(* Logix 5000 project; controller reports 1756-L63 rev 20.11; software revision 20.04; part 40 of 52 *)

        [82].log_data[53].total := -6932.722, [82].log_data[53].time := 3600.0, [82].log_data[53].minminute := 24, [82].log_data[53].maxminute := 3, [82].log_data[53].valid := 1, [82].log_data[54].max := 0.5155, [82].log_data[54].total := 1254.2913, [82].log_data[54].time := 3600.0, [82].log_data[54].minminute := 8, [82].log_data[54].maxminute := 9, [82].log_data[54].valid := 1, [82].log_data[55].max := 0.52349997, [82].log_data[55].total := 1217.507, [82].log_data[55].time := 3600.0, [82].log_data[55].minminute := 1, [82].log_data[55].maxminute := 24, [82].log_data[55].valid := 1, [82].log_data[56].min := 0.159696, [82].log_data[56].max := 0.16024561, [82].log_data[56].total := 575.79816, [82].log_data[56].time := 3600.0, [82].log_data[56].minminute := 6, [82].log_data[56].maxminute := 3, [82].log_data[56].valid := 1, [82].log_data[57].min := 0.24818413, [82].log_data[57].max := 0.2500293, [82].log_data[57].total := 894.9429, [82].log_data[57].time := 3600.0, [82].log_data[57].minminute := 17, [82].log_data[57].maxminute := 1, [82].log_data[57].valid := 1, [82].log_data[58].time := 3600.0, [82].log_data[58].valid := 1, [82].log_data[59].time := 3600.0, [82].log_data[59].valid := 1, [82].log_data[60].valid := 1, [82].log_data[61].valid := 1, [82].log_data[62].valid := 1, [82].log_data[63].valid := 1, [82].log_data[64].valid := 1, [82].log_data[65].valid := 1, [82].log_data[66].valid := 1, [82].log_data[67].valid := 1, [82].log_data[68].valid := 1, [82].log_data[69].valid := 1, [82].log_data[70].valid := 1, [82].log_data[71].valid := 1, [82].log_data[72].valid := 1, [82].log_data[73].valid := 1, [82].log_data[74].valid := 1, [82].log_data[75].valid := 1, [82].log_data[76].valid := 1, [82].log_data[77].valid := 1, [82].log_data[78].valid := 1, [82].log_data[79].valid := 1, [82].log_data[80].valid := 1, [82].log_data[81].valid := 1, [82].log_data[82].valid := 1, [82].log_data[83].valid := 1, [82].log_data[84].valid := 1,
        [82].log_data[85].valid := 1, [82].log_data[86].valid := 1, [82].log_data[87].valid := 1, [82].log_data[88].valid := 1, [82].log_data[89].valid := 1, [82].log_data[90].valid := 1, [82].log_data[91].valid := 1, [82].log_data[92].valid := 1, [82].log_data[93].valid := 1, [82].log_data[94].valid := 1, [82].log_data[95].valid := 1, [82].log_data[96].valid := 1, [82].log_data[97].valid := 1, [82].log_data[98].valid := 1, [82].log_data[99].valid := 1, [82].log_data[100].valid := 1, [82].log_data[101].valid := 1, [82].log_data[102].valid := 1, [82].log_data[103].valid := 1, [82].log_data[104].valid := 1, [82].log_data[105].valid := 1, [82].log_data[106].valid := 1, [82].log_data[107].valid := 1, [82].log_data[108].valid := 1, [82].log_data[109].valid := 1, [82].log_data[110].valid := 1, [82].log_data[111].valid := 1, [82].log_data[112].valid := 1, [82].log_data[113].valid := 1, [82].log_data[114].valid := 1, [82].log_data[115].valid := 1, [82].log_data[116].valid := 1, [82].log_data[117].valid := 1, [82].log_data[118].valid := 1, [82].log_data[119].valid := 1, [82].log_data[120].valid := 1, [82].log_data[121].valid := 1, [82].log_data[122].valid := 1, [82].log_data[123].valid := 1, [82].log_data[124].valid := 1, [82].time.Year := 2023, [82].time.Month := 1, [82].time.Day := 16, [82].time.Hour := 13, [82].time.Minute := 59, [82].time.Second := 59, [83].log_data[0].min := 1.0, [83].log_data[0].max := 1.0, [83].log_data[0].total := 3600.0, [83].log_data[0].time := 3600.0, [83].log_data[0].valid := 1, [83].log_data[1].max := 1.0, [83].log_data[1].total := 542.0, [83].log_data[1].time := 3600.0, [83].log_data[1].maxminute := 41, [83].log_data[1].valid := 1, [83].log_data[2].max := 1.0, [83].log_data[2].total := 538.5, [83].log_data[2].time := 3600.0, [83].log_data[2].maxminute := 41,
        [83].log_data[2].valid := 1, [83].log_data[3].time := 3600.0, [83].log_data[3].valid := 1, [83].log_data[4].time := 3600.0, [83].log_data[4].valid := 1, [83].log_data[5].max := 1.0, [83].log_data[5].total := 231.0, [83].log_data[5].time := 3600.0, [83].log_data[5].maxminute := 44, [83].log_data[5].valid := 1, [83].log_data[6].time := 3600.0, [83].log_data[6].valid := 1, [83].log_data[7].time := 3600.0, [83].log_data[7].valid := 1, [83].log_data[8].max := 1.0, [83].log_data[8].total := 1310.5, [83].log_data[8].time := 3600.0, [83].log_data[8].minminute := 10, [83].log_data[8].valid := 1, [83].log_data[9].max := 1.0, [83].log_data[9].total := 1307.0, [83].log_data[9].time := 3600.0, [83].log_data[9].minminute := 10, [83].log_data[9].valid := 1, [83].log_data[10].min := 1.0, [83].log_data[10].max := 1.0, [83].log_data[10].total := 3600.0, [83].log_data[10].time := 3600.0, [83].log_data[10].valid := 1, [83].log_data[11].time := 3600.0, [83].log_data[11].valid := 1, [83].log_data[12].min := 1.0, [83].log_data[12].max := 1.0, [83].log_data[12].total := 3600.0, [83].log_data[12].time := 3600.0, [83].log_data[12].valid := 1, [83].log_data[13].min := 1.0, [83].log_data[13].max := 1.0, [83].log_data[13].total := 3600.0, [83].log_data[13].time := 3600.0, [83].log_data[13].valid := 1, [83].log_data[14].time := 3600.0, [83].log_data[14].valid := 1, [83].log_data[15].time := 3600.0, [83].log_data[15].valid := 1, [83].log_data[16].time := 3600.0, [83].log_data[16].valid := 1, [83].log_data[17].min := 1.0, [83].log_data[17].max := 1.0, [83].log_data[17].total := 3600.0, [83].log_data[17].time := 3600.0, [83].log_data[17].valid := 1, [83].log_data[18].time := 3600.0, [83].log_data[18].valid := 1, [83].log_data[19].time := 3600.0, [83].log_data[19].valid := 1, [83].log_data[20].time := 3600.0, [83].log_data[20].valid := 1, [83].log_data[21].min := 1.0, [83].log_data[21].max := 1.0,
        [83].log_data[21].total := 3600.0, [83].log_data[21].time := 3600.0, [83].log_data[21].valid := 1, [83].log_data[22].time := 3600.0, [83].log_data[22].valid := 1, [83].log_data[23].time := 3600.0, [83].log_data[23].valid := 1, [83].log_data[24].time := 3600.0, [83].log_data[24].valid := 1, [83].log_data[25].time := 3600.0, [83].log_data[25].valid := 1, [83].log_data[26].time := 3600.0, [83].log_data[26].valid := 1, [83].log_data[27].time := 3600.0, [83].log_data[27].valid := 1, [83].log_data[28].time := 3600.0, [83].log_data[28].valid := 1, [83].log_data[29].min := 1.0, [83].log_data[29].max := 1.0, [83].log_data[29].total := 3600.0, [83].log_data[29].time := 3600.0, [83].log_data[29].valid := 1, [83].log_data[30].min := 1.0, [83].log_data[30].max := 1.0, [83].log_data[30].total := 3600.0, [83].log_data[30].time := 3600.0, [83].log_data[30].valid := 1, [83].log_data[31].max := 1.0, [83].log_data[31].total := 1071.998, [83].log_data[31].time := 3600.0, [83].log_data[31].maxminute := 2, [83].log_data[31].valid := 1, [83].log_data[32].max := 1.0, [83].log_data[32].total := 57.749, [83].log_data[32].time := 3600.0, [83].log_data[32].valid := 1, [83].log_data[33].max := 1.0, [83].log_data[33].total := 974.5, [83].log_data[33].time := 3600.0, [83].log_data[33].maxminute := 10, [83].log_data[33].valid := 1, [83].log_data[34].max := 1.0, [83].log_data[34].total := 987.5, [83].log_data[34].time := 3600.0, [83].log_data[34].maxminute := 8, [83].log_data[34].valid := 1, [83].log_data[35].max := 1.0, [83].log_data[35].total := 538.998, [83].log_data[35].time := 3600.0, [83].log_data[35].maxminute := 6, [83].log_data[35].valid := 1, [83].log_data[36].max := 1.0, [83].log_data[36].total := 571.5, [83].log_data[36].time := 3600.0, [83].log_data[36].minminute := 5, [83].log_data[36].valid := 1, [83].log_data[37].max := 7.3565416, [83].log_data[37].total := 3456.338, [83].log_data[37].time := 3600.0, [83].log_data[37].maxminute := 44,
        [83].log_data[37].valid := 1, [83].log_data[38].time := 3600.0, [83].log_data[38].valid := 1, [83].log_data[39].min := 0.994824, [83].log_data[39].max := 1.0214411, [83].log_data[39].total := 3605.966, [83].log_data[39].time := 3600.0, [83].log_data[39].minminute := 3, [83].log_data[39].maxminute := 48, [83].log_data[39].valid := 1, [83].log_data[40].min := 7.574485, [83].log_data[40].max := 7.60224, [83].log_data[40].total := 27337.104, [83].log_data[40].time := 3600.0, [83].log_data[40].minminute := 29, [83].log_data[40].maxminute := 32, [83].log_data[40].valid := 1, [83].log_data[41].min := 0.02273633, [83].log_data[41].max := 0.035495363, [83].log_data[41].total := 89.72992, [83].log_data[41].time := 3600.0, [83].log_data[41].minminute := 20, [83].log_data[41].maxminute := 32, [83].log_data[41].valid := 1, [83].log_data[42].min := 2.291407, [83].log_data[42].max := 2.2964714, [83].log_data[42].total := 8258.98, [83].log_data[42].time := 3600.0, [83].log_data[42].minminute := 56, [83].log_data[42].maxminute := 28, [83].log_data[42].valid := 1, [83].log_data[43].min := -0.27999878, [83].log_data[43].max := -0.26000214, [83].log_data[43].total := -981.76685, [83].log_data[43].time := 3600.0, [83].log_data[43].maxminute := 2, [83].log_data[43].valid := 1, [83].log_data[44].min := -0.3199997, [83].log_data[44].max := -0.30000305, [83].log_data[44].total := -1089.0538, [83].log_data[44].time := 3600.0, [83].log_data[44].valid := 1, [83].log_data[45].time := 3600.0, [83].log_data[45].valid := 1, [83].log_data[46].time := 3600.0, [83].log_data[46].valid := 1, [83].log_data[47].time := 3600.0, [83].log_data[47].valid := 1, [83].log_data[48].min := 6.7179084, [83].log_data[48].max := 6.9322586, [83].log_data[48].total := 24380.49, [83].log_data[48].time := 3600.0, [83].log_data[48].minminute := 59, [83].log_data[48].maxminute := 50, [83].log_data[48].valid := 1, [83].log_data[49].min := 7.303773, [83].log_data[49].max := 9.598419, [83].log_data[49].total := 33269.867, [83].log_data[49].time := 3600.0, [83].log_data[49].minminute := 59,
        [83].log_data[49].maxminute := 5, [83].log_data[49].valid := 1, [83].log_data[50].min := 1.9989722, [83].log_data[50].max := 2.151373, [83].log_data[50].total := 7406.148, [83].log_data[50].time := 3600.0, [83].log_data[50].minminute := 10, [83].log_data[50].maxminute := 49, [83].log_data[50].valid := 1, [83].log_data[51].max := 3.127, [83].log_data[51].total := 2959.4797, [83].log_data[51].time := 3600.0, [83].log_data[51].maxminute := 10, [83].log_data[51].valid := 1, [83].log_data[52].min := -5.739998, [83].log_data[52].max := 0.11999512, [83].log_data[52].total := -8463.669, [83].log_data[52].time := 3600.0, [83].log_data[52].minminute := 49, [83].log_data[52].valid := 1, [83].log_data[53].min := -4.919998, [83].log_data[53].max := 0.30000305, [83].log_data[53].total := -7675.482, [83].log_data[53].time := 3600.0, [83].log_data[53].minminute := 49, [83].log_data[53].maxminute := 55, [83].log_data[53].valid := 1, [83].log_data[54].max := 0.56850004, [83].log_data[54].total := 446.67337, [83].log_data[54].time := 3600.0, [83].log_data[54].maxminute := 2, [83].log_data[54].valid := 1, [83].log_data[55].max := 0.543, [83].log_data[55].total := 438.6968, [83].log_data[55].time := 3600.0, [83].log_data[55].minminute := 5, [83].log_data[55].maxminute := 55, [83].log_data[55].valid := 1, [83].log_data[56].min := 0.15973525, [83].log_data[56].max := 0.16016708, [83].log_data[56].total := 575.74774, [83].log_data[56].time := 3600.0, [83].log_data[56].minminute := 12, [83].log_data[56].maxminute := 17, [83].log_data[56].valid := 1, [83].log_data[57].min := 0.24818413, [83].log_data[57].max := 0.24861601, [83].log_data[57].total := 894.0131, [83].log_data[57].time := 3600.0, [83].log_data[57].maxminute := 39, [83].log_data[57].valid := 1, [83].log_data[58].time := 3600.0, [83].log_data[58].valid := 1, [83].log_data[59].time := 3600.0, [83].log_data[59].valid := 1, [83].log_data[60].valid := 1, [83].log_data[61].valid := 1, [83].log_data[62].valid := 1, [83].log_data[63].valid := 1, [83].log_data[64].valid := 1,
        [83].log_data[65].valid := 1, [83].log_data[66].valid := 1, [83].log_data[67].valid := 1, [83].log_data[68].valid := 1, [83].log_data[69].valid := 1, [83].log_data[70].valid := 1, [83].log_data[71].valid := 1, [83].log_data[72].valid := 1, [83].log_data[73].valid := 1, [83].log_data[74].valid := 1, [83].log_data[75].valid := 1, [83].log_data[76].valid := 1, [83].log_data[77].valid := 1, [83].log_data[78].valid := 1, [83].log_data[79].valid := 1, [83].log_data[80].valid := 1, [83].log_data[81].valid := 1, [83].log_data[82].valid := 1, [83].log_data[83].valid := 1, [83].log_data[84].valid := 1, [83].log_data[85].valid := 1, [83].log_data[86].valid := 1, [83].log_data[87].valid := 1, [83].log_data[88].valid := 1, [83].log_data[89].valid := 1, [83].log_data[90].valid := 1, [83].log_data[91].valid := 1, [83].log_data[92].valid := 1, [83].log_data[93].valid := 1, [83].log_data[94].valid := 1, [83].log_data[95].valid := 1, [83].log_data[96].valid := 1, [83].log_data[97].valid := 1, [83].log_data[98].valid := 1, [83].log_data[99].valid := 1, [83].log_data[100].valid := 1, [83].log_data[101].valid := 1, [83].log_data[102].valid := 1, [83].log_data[103].valid := 1, [83].log_data[104].valid := 1, [83].log_data[105].valid := 1, [83].log_data[106].valid := 1, [83].log_data[107].valid := 1, [83].log_data[108].valid := 1, [83].log_data[109].valid := 1, [83].log_data[110].valid := 1, [83].log_data[111].valid := 1, [83].log_data[112].valid := 1, [83].log_data[113].valid := 1, [83].log_data[114].valid := 1, [83].log_data[115].valid := 1, [83].log_data[116].valid := 1, [83].log_data[117].valid := 1, [83].log_data[118].valid := 1, [83].log_data[119].valid := 1, [83].log_data[120].valid := 1, [83].log_data[121].valid := 1, [83].log_data[122].valid := 1, [83].log_data[123].valid := 1, [83].log_data[124].valid := 1,
        [83].time.Year := 2023, [83].time.Month := 1, [83].time.Day := 16, [83].time.Hour := 14, [83].time.Minute := 59, [83].time.Second := 59, [84].log_data[0].min := 1.0, [84].log_data[0].max := 1.0, [84].log_data[0].total := 3600.0, [84].log_data[0].time := 3600.0, [84].log_data[0].valid := 1, [84].log_data[1].time := 3600.0, [84].log_data[1].valid := 1, [84].log_data[2].time := 3600.0, [84].log_data[2].valid := 1, [84].log_data[3].time := 3600.0, [84].log_data[3].valid := 1, [84].log_data[4].time := 3600.0, [84].log_data[4].valid := 1, [84].log_data[5].time := 3600.0, [84].log_data[5].valid := 1, [84].log_data[6].time := 3600.0, [84].log_data[6].valid := 1, [84].log_data[7].time := 3600.0, [84].log_data[7].valid := 1, [84].log_data[8].max := 1.0, [84].log_data[8].total := 322.251, [84].log_data[8].time := 3600.0, [84].log_data[8].minminute := 5, [84].log_data[8].valid := 1, [84].log_data[9].max := 1.0, [84].log_data[9].total := 322.251, [84].log_data[9].time := 3600.0, [84].log_data[9].minminute := 5, [84].log_data[9].valid := 1, [84].log_data[10].min := 1.0, [84].log_data[10].max := 1.0, [84].log_data[10].total := 3600.0, [84].log_data[10].time := 3600.0, [84].log_data[10].valid := 1, [84].log_data[11].time := 3600.0, [84].log_data[11].valid := 1, [84].log_data[12].min := 1.0, [84].log_data[12].max := 1.0, [84].log_data[12].total := 3600.0, [84].log_data[12].time := 3600.0, [84].log_data[12].valid := 1, [84].log_data[13].min := 1.0, [84].log_data[13].max := 1.0, [84].log_data[13].total := 3600.0, [84].log_data[13].time := 3600.0, [84].log_data[13].valid := 1, [84].log_data[14].time := 3600.0, [84].log_data[14].valid := 1, [84].log_data[15].time := 3600.0, [84].log_data[15].valid := 1, [84].log_data[16].time := 3600.0, [84].log_data[16].valid := 1, [84].log_data[17].min := 1.0, [84].log_data[17].max := 1.0,
        [84].log_data[17].total := 3600.0, [84].log_data[17].time := 3600.0, [84].log_data[17].valid := 1, [84].log_data[18].time := 3600.0, [84].log_data[18].valid := 1, [84].log_data[19].time := 3600.0, [84].log_data[19].valid := 1, [84].log_data[20].time := 3600.0, [84].log_data[20].valid := 1, [84].log_data[21].min := 1.0, [84].log_data[21].max := 1.0, [84].log_data[21].total := 3600.0, [84].log_data[21].time := 3600.0, [84].log_data[21].valid := 1, [84].log_data[22].time := 3600.0, [84].log_data[22].valid := 1, [84].log_data[23].time := 3600.0, [84].log_data[23].valid := 1, [84].log_data[24].time := 3600.0, [84].log_data[24].valid := 1, [84].log_data[25].time := 3600.0, [84].log_data[25].valid := 1, [84].log_data[26].time := 3600.0, [84].log_data[26].valid := 1, [84].log_data[27].time := 3600.0, [84].log_data[27].valid := 1, [84].log_data[28].time := 3600.0, [84].log_data[28].valid := 1, [84].log_data[29].min := 1.0, [84].log_data[29].max := 1.0, [84].log_data[29].total := 3600.0, [84].log_data[29].time := 3600.0, [84].log_data[29].valid := 1, [84].log_data[30].min := 1.0, [84].log_data[30].max := 1.0, [84].log_data[30].total := 3600.0, [84].log_data[30].time := 3600.0, [84].log_data[30].valid := 1, [84].log_data[31].time := 3600.0, [84].log_data[31].valid := 1, [84].log_data[32].max := 1.0, [84].log_data[32].total := 238.749, [84].log_data[32].time := 3600.0, [84].log_data[32].maxminute := 1, [84].log_data[32].valid := 1, [84].log_data[33].time := 3600.0, [84].log_data[33].valid := 1, [84].log_data[34].time := 3600.0, [84].log_data[34].valid := 1, [84].log_data[35].max := 1.0, [84].log_data[35].total := 276.0, [84].log_data[35].time := 3600.0, [84].log_data[35].minminute := 4, [84].log_data[35].valid := 1, [84].log_data[36].time := 3600.0, [84].log_data[36].valid := 1, [84].log_data[37].time := 3600.0, [84].log_data[37].valid := 1, [84].log_data[38].time := 3600.0, [84].log_data[38].valid := 1,
        [84].log_data[39].min := 0.99494183, [84].log_data[39].max := 1.0055416, [84].log_data[39].total := 3602.3838, [84].log_data[39].time := 3600.0, [84].log_data[39].minminute := 16, [84].log_data[39].maxminute := 46, [84].log_data[39].valid := 1, [84].log_data[40].min := 7.5816298, [84].log_data[40].max := 7.604989, [84].log_data[40].total := 27343.059, [84].log_data[40].time := 3600.0, [84].log_data[40].minminute := 26, [84].log_data[40].maxminute := 37, [84].log_data[40].valid := 1, [84].log_data[41].min := 0.02273633, [84].log_data[41].max := 0.030195557, [84].log_data[41].total := 87.1149, [84].log_data[41].time := 3600.0, [84].log_data[41].minminute := 1, [84].log_data[41].maxminute := 57, [84].log_data[41].valid := 1, [84].log_data[42].min := 2.291525, [84].log_data[42].max := 2.2963536, [84].log_data[42].total := 8259.134, [84].log_data[42].time := 3600.0, [84].log_data[42].minminute := 10, [84].log_data[42].maxminute := 47, [84].log_data[42].valid := 1, [84].log_data[43].min := -0.27999878, [84].log_data[43].max := -0.26000214, [84].log_data[43].total := -936.00824, [84].log_data[43].time := 3600.0, [84].log_data[43].valid := 1, [84].log_data[44].min := -0.30000305, [84].log_data[44].max := -0.27999878, [84].log_data[44].total := -1061.0931, [84].log_data[44].time := 3600.0, [84].log_data[44].maxminute := 5, [84].log_data[44].valid := 1, [84].log_data[45].time := 3600.0, [84].log_data[45].valid := 1, [84].log_data[46].time := 3600.0, [84].log_data[46].valid := 1, [84].log_data[47].time := 3600.0, [84].log_data[47].valid := 1, [84].log_data[48].min := 6.5678625, [84].log_data[48].max := 6.7181826, [84].log_data[48].total := 23808.375, [84].log_data[48].time := 3600.0, [84].log_data[48].minminute := 18, [84].log_data[48].valid := 1, [84].log_data[49].min := 6.593787, [84].log_data[49].max := 9.412138, [84].log_data[49].total := 28587.87, [84].log_data[49].time := 3600.0, [84].log_data[49].minminute := 17, [84].log_data[49].maxminute := 59, [84].log_data[49].valid := 1, [84].log_data[50].min := 1.9986188, [84].log_data[50].max := 2.109445,
        [84].log_data[50].total := 7530.9287, [84].log_data[50].time := 3600.0, [84].log_data[50].minminute := 5, [84].log_data[50].maxminute := 57, [84].log_data[50].valid := 1, [84].log_data[51].time := 3600.0, [84].log_data[51].valid := 1, [84].log_data[52].min := -2.9199982, [84].log_data[52].max := 0.11999512, [84].log_data[52].total := -5281.0723, [84].log_data[52].time := 3600.0, [84].log_data[52].minminute := 1, [84].log_data[52].valid := 1, [84].log_data[53].min := -2.4000015, [84].log_data[53].max := 0.22000122, [84].log_data[53].total := -5018.0986, [84].log_data[53].time := 3600.0, [84].log_data[53].minminute := 4, [84].log_data[53].maxminute := 5, [84].log_data[53].valid := 1, [84].log_data[54].max := 0.523, [84].log_data[54].total := 93.84478, [84].log_data[54].time := 3600.0, [84].log_data[54].maxminute := 1, [84].log_data[54].valid := 1, [84].log_data[55].max := 0.4465, [84].log_data[55].total := 110.74925, [84].log_data[55].time := 3600.0, [84].log_data[55].minminute := 4, [84].log_data[55].maxminute := 4, [84].log_data[55].valid := 1, [84].log_data[56].min := 0.15973525, [84].log_data[56].max := 0.16012783, [84].log_data[56].total := 575.5827, [84].log_data[56].time := 3600.0, [84].log_data[56].minminute := 19, [84].log_data[56].maxminute := 1, [84].log_data[56].valid := 1, [84].log_data[57].min := 0.24826264, [84].log_data[57].max := 0.24869452, [84].log_data[57].total := 894.43835, [84].log_data[57].time := 3600.0, [84].log_data[57].minminute := 23, [84].log_data[57].maxminute := 37, [84].log_data[57].valid := 1, [84].log_data[58].time := 3600.0, [84].log_data[58].valid := 1, [84].log_data[59].time := 3600.0, [84].log_data[59].valid := 1, [84].log_data[60].valid := 1, [84].log_data[61].valid := 1, [84].log_data[62].valid := 1, [84].log_data[63].valid := 1, [84].log_data[64].valid := 1, [84].log_data[65].valid := 1, [84].log_data[66].valid := 1, [84].log_data[67].valid := 1, [84].log_data[68].valid := 1, [84].log_data[69].valid := 1, [84].log_data[70].valid := 1,
        [84].log_data[71].valid := 1, [84].log_data[72].valid := 1, [84].log_data[73].valid := 1, [84].log_data[74].valid := 1, [84].log_data[75].valid := 1, [84].log_data[76].valid := 1, [84].log_data[77].valid := 1, [84].log_data[78].valid := 1, [84].log_data[79].valid := 1, [84].log_data[80].valid := 1, [84].log_data[81].valid := 1, [84].log_data[82].valid := 1, [84].log_data[83].valid := 1, [84].log_data[84].valid := 1, [84].log_data[85].valid := 1, [84].log_data[86].valid := 1, [84].log_data[87].valid := 1, [84].log_data[88].valid := 1, [84].log_data[89].valid := 1, [84].log_data[90].valid := 1, [84].log_data[91].valid := 1, [84].log_data[92].valid := 1, [84].log_data[93].valid := 1, [84].log_data[94].valid := 1, [84].log_data[95].valid := 1, [84].log_data[96].valid := 1, [84].log_data[97].valid := 1, [84].log_data[98].valid := 1, [84].log_data[99].valid := 1, [84].log_data[100].valid := 1, [84].log_data[101].valid := 1, [84].log_data[102].valid := 1, [84].log_data[103].valid := 1, [84].log_data[104].valid := 1, [84].log_data[105].valid := 1, [84].log_data[106].valid := 1, [84].log_data[107].valid := 1, [84].log_data[108].valid := 1, [84].log_data[109].valid := 1, [84].log_data[110].valid := 1, [84].log_data[111].valid := 1, [84].log_data[112].valid := 1, [84].log_data[113].valid := 1, [84].log_data[114].valid := 1, [84].log_data[115].valid := 1, [84].log_data[116].valid := 1, [84].log_data[117].valid := 1, [84].log_data[118].valid := 1, [84].log_data[119].valid := 1, [84].log_data[120].valid := 1, [84].log_data[121].valid := 1, [84].log_data[122].valid := 1, [84].log_data[123].valid := 1, [84].log_data[124].valid := 1, [84].time.Year := 2023, [84].time.Month := 1, [84].time.Day := 16, [84].time.Hour := 15, [84].time.Minute := 59, [84].time.Second := 59,
        [85].log_data[0].min := 1.0, [85].log_data[0].max := 1.0, [85].log_data[0].total := 3600.0, [85].log_data[0].time := 3600.0, [85].log_data[0].valid := 1, [85].log_data[1].max := 1.0, [85].log_data[1].total := 541.5, [85].log_data[1].time := 3600.0, [85].log_data[1].maxminute := 47, [85].log_data[1].valid := 1, [85].log_data[2].max := 1.0, [85].log_data[2].total := 538.0, [85].log_data[2].time := 3600.0, [85].log_data[2].maxminute := 47, [85].log_data[2].valid := 1, [85].log_data[3].time := 3600.0, [85].log_data[3].valid := 1, [85].log_data[4].time := 3600.0, [85].log_data[4].valid := 1, [85].log_data[5].max := 1.0, [85].log_data[5].total := 244.5, [85].log_data[5].time := 3600.0, [85].log_data[5].maxminute := 49, [85].log_data[5].valid := 1, [85].log_data[6].time := 3600.0, [85].log_data[6].valid := 1, [85].log_data[7].time := 3600.0, [85].log_data[7].valid := 1, [85].log_data[8].max := 1.0, [85].log_data[8].total := 508.749, [85].log_data[8].time := 3600.0, [85].log_data[8].maxminute := 51, [85].log_data[8].valid := 1, [85].log_data[9].max := 1.0, [85].log_data[9].total := 505.249, [85].log_data[9].time := 3600.0, [85].log_data[9].maxminute := 51, [85].log_data[9].valid := 1, [85].log_data[10].min := 1.0, [85].log_data[10].max := 1.0, [85].log_data[10].total := 3600.0, [85].log_data[10].time := 3600.0, [85].log_data[10].valid := 1, [85].log_data[11].time := 3600.0, [85].log_data[11].valid := 1, [85].log_data[12].min := 1.0, [85].log_data[12].max := 1.0, [85].log_data[12].total := 3600.0, [85].log_data[12].time := 3600.0, [85].log_data[12].valid := 1, [85].log_data[13].min := 1.0, [85].log_data[13].max := 1.0, [85].log_data[13].total := 3600.0, [85].log_data[13].time := 3600.0, [85].log_data[13].valid := 1, [85].log_data[14].time := 3600.0, [85].log_data[14].valid := 1, [85].log_data[15].time := 3600.0, [85].log_data[15].valid := 1, [85].log_data[16].time := 3600.0,
        [85].log_data[16].valid := 1, [85].log_data[17].min := 1.0, [85].log_data[17].max := 1.0, [85].log_data[17].total := 3600.0, [85].log_data[17].time := 3600.0, [85].log_data[17].valid := 1, [85].log_data[18].time := 3600.0, [85].log_data[18].valid := 1, [85].log_data[19].time := 3600.0, [85].log_data[19].valid := 1, [85].log_data[20].time := 3600.0, [85].log_data[20].valid := 1, [85].log_data[21].min := 1.0, [85].log_data[21].max := 1.0, [85].log_data[21].total := 3600.0, [85].log_data[21].time := 3600.0, [85].log_data[21].valid := 1, [85].log_data[22].time := 3600.0, [85].log_data[22].valid := 1, [85].log_data[23].time := 3600.0, [85].log_data[23].valid := 1, [85].log_data[24].time := 3600.0, [85].log_data[24].valid := 1, [85].log_data[25].time := 3600.0, [85].log_data[25].valid := 1, [85].log_data[26].time := 3600.0, [85].log_data[26].valid := 1, [85].log_data[27].time := 3600.0, [85].log_data[27].valid := 1, [85].log_data[28].time := 3600.0, [85].log_data[28].valid := 1, [85].log_data[29].min := 1.0, [85].log_data[29].max := 1.0, [85].log_data[29].total := 3600.0, [85].log_data[29].time := 3600.0, [85].log_data[29].valid := 1, [85].log_data[30].min := 1.0, [85].log_data[30].max := 1.0, [85].log_data[30].total := 3600.0, [85].log_data[30].time := 3600.0, [85].log_data[30].valid := 1, [85].log_data[31].max := 1.0, [85].log_data[31].total := 304.249, [85].log_data[31].time := 3600.0, [85].log_data[31].maxminute := 51, [85].log_data[31].valid := 1, [85].log_data[32].max := 1.0, [85].log_data[32].total := 109.249, [85].log_data[32].time := 3600.0, [85].log_data[32].maxminute := 58, [85].log_data[32].valid := 1, [85].log_data[33].time := 3600.0, [85].log_data[33].valid := 1, [85].log_data[34].time := 3600.0, [85].log_data[34].valid := 1, [85].log_data[35].time := 3600.0, [85].log_data[35].valid := 1, [85].log_data[36].max := 1.0, [85].log_data[36].total := 498.249, [85].log_data[36].time := 3600.0,
        [85].log_data[36].maxminute := 51, [85].log_data[36].valid := 1, [85].log_data[37].max := 7.6030836, [85].log_data[37].total := 3563.115, [85].log_data[37].time := 3600.0, [85].log_data[37].maxminute := 49, [85].log_data[37].valid := 1, [85].log_data[38].time := 3600.0, [85].log_data[38].valid := 1, [85].log_data[39].min := 0.994824, [85].log_data[39].max := 1.0213233, [85].log_data[39].total := 3607.2905, [85].log_data[39].time := 3600.0, [85].log_data[39].minminute := 13, [85].log_data[39].maxminute := 54, [85].log_data[39].valid := 1, [85].log_data[40].min := 7.5802555, [85].log_data[40].max := 7.603339, [85].log_data[40].total := 27341.73, [85].log_data[40].time := 3600.0, [85].log_data[40].minminute := 26, [85].log_data[40].maxminute := 31, [85].log_data[40].valid := 1, [85].log_data[41].min := 0.02273633, [85].log_data[41].max := 0.036476806, [85].log_data[41].total := 93.75936, [85].log_data[41].time := 3600.0, [85].log_data[41].minminute := 19, [85].log_data[41].maxminute := 12, [85].log_data[41].valid := 1, [85].log_data[42].min := 2.291525, [85].log_data[42].max := 2.2964714, [85].log_data[42].total := 8259.261, [85].log_data[42].time := 3600.0, [85].log_data[42].minminute := 7, [85].log_data[42].maxminute := 41, [85].log_data[42].valid := 1, [85].log_data[43].min := -0.26000214, [85].log_data[43].max := -0.23999786, [85].log_data[43].total := -935.90826, [85].log_data[43].time := 3600.0, [85].log_data[43].maxminute := 1, [85].log_data[43].valid := 1, [85].log_data[44].min := -0.30000305, [85].log_data[44].max := -0.27999878, [85].log_data[44].total := -1013.5552, [85].log_data[44].time := 3600.0, [85].log_data[44].valid := 1, [85].log_data[45].time := 3600.0, [85].log_data[45].valid := 1, [85].log_data[46].time := 3600.0, [85].log_data[46].valid := 1, [85].log_data[47].time := 3600.0, [85].log_data[47].valid := 1, [85].log_data[48].min := 6.6335416, [85].log_data[48].max := 6.9078, [85].log_data[48].total := 24063.035, [85].log_data[48].time := 3600.0, [85].log_data[48].maxminute := 56, [85].log_data[48].valid := 1,
        [85].log_data[49].min := 8.170596, [85].log_data[49].max := 9.692444, [85].log_data[49].total := 34133.863, [85].log_data[49].time := 3600.0, [85].log_data[49].minminute := 59, [85].log_data[49].maxminute := 49, [85].log_data[49].valid := 1, [85].log_data[50].min := 2.0683415, [85].log_data[50].max := 2.1509018, [85].log_data[50].total := 7587.8726, [85].log_data[50].time := 3600.0, [85].log_data[50].minminute := 54, [85].log_data[50].maxminute := 51, [85].log_data[50].valid := 1, [85].log_data[51].time := 3600.0, [85].log_data[51].valid := 1, [85].log_data[52].min := -4.3199997, [85].log_data[52].max := 0.11999512, [85].log_data[52].total := -5856.0786, [85].log_data[52].time := 3600.0, [85].log_data[52].minminute := 51, [85].log_data[52].maxminute := 56, [85].log_data[52].valid := 1, [85].log_data[53].min := -4.040001, [85].log_data[53].max := -1.4400024, [85].log_data[53].total := -5783.3413, [85].log_data[53].time := 3600.0, [85].log_data[53].minminute := 51, [85].log_data[53].valid := 1, [85].log_data[54].max := 0.508, [85].log_data[54].total := 161.4602, [85].log_data[54].time := 3600.0, [85].log_data[54].maxminute := 51, [85].log_data[54].valid := 1, [85].log_data[55].max := 0.5005, [85].log_data[55].total := 197.12991, [85].log_data[55].time := 3600.0, [85].log_data[55].maxminute := 51, [85].log_data[55].valid := 1, [85].log_data[56].min := 0.15961748, [85].log_data[56].max := 0.16012783, [85].log_data[56].total := 575.4132, [85].log_data[56].time := 3600.0, [85].log_data[56].minminute := 45, [85].log_data[56].maxminute := 49, [85].log_data[56].valid := 1, [85].log_data[57].min := 0.24838047, [85].log_data[57].max := 0.2488123, [85].log_data[57].total := 894.79694, [85].log_data[57].time := 3600.0, [85].log_data[57].minminute := 3, [85].log_data[57].maxminute := 25, [85].log_data[57].valid := 1, [85].log_data[58].time := 3600.0, [85].log_data[58].valid := 1, [85].log_data[59].time := 3600.0, [85].log_data[59].valid := 1, [85].log_data[60].valid := 1, [85].log_data[61].valid := 1, [85].log_data[62].valid := 1,
        [85].log_data[63].valid := 1, [85].log_data[64].valid := 1, [85].log_data[65].valid := 1, [85].log_data[66].valid := 1, [85].log_data[67].valid := 1, [85].log_data[68].valid := 1, [85].log_data[69].valid := 1, [85].log_data[70].valid := 1, [85].log_data[71].valid := 1, [85].log_data[72].valid := 1, [85].log_data[73].valid := 1, [85].log_data[74].valid := 1, [85].log_data[75].valid := 1, [85].log_data[76].valid := 1, [85].log_data[77].valid := 1, [85].log_data[78].valid := 1, [85].log_data[79].valid := 1, [85].log_data[80].valid := 1, [85].log_data[81].valid := 1, [85].log_data[82].valid := 1, [85].log_data[83].valid := 1, [85].log_data[84].valid := 1, [85].log_data[85].valid := 1, [85].log_data[86].valid := 1, [85].log_data[87].valid := 1, [85].log_data[88].valid := 1, [85].log_data[89].valid := 1, [85].log_data[90].valid := 1, [85].log_data[91].valid := 1, [85].log_data[92].valid := 1, [85].log_data[93].valid := 1, [85].log_data[94].valid := 1, [85].log_data[95].valid := 1, [85].log_data[96].valid := 1, [85].log_data[97].valid := 1, [85].log_data[98].valid := 1, [85].log_data[99].valid := 1, [85].log_data[100].valid := 1, [85].log_data[101].valid := 1, [85].log_data[102].valid := 1, [85].log_data[103].valid := 1, [85].log_data[104].valid := 1, [85].log_data[105].valid := 1, [85].log_data[106].valid := 1, [85].log_data[107].valid := 1, [85].log_data[108].valid := 1, [85].log_data[109].valid := 1, [85].log_data[110].valid := 1, [85].log_data[111].valid := 1, [85].log_data[112].valid := 1, [85].log_data[113].valid := 1, [85].log_data[114].valid := 1, [85].log_data[115].valid := 1, [85].log_data[116].valid := 1, [85].log_data[117].valid := 1, [85].log_data[118].valid := 1, [85].log_data[119].valid := 1, [85].log_data[120].valid := 1, [85].log_data[121].valid := 1, [85].log_data[122].valid := 1,
        [85].log_data[123].valid := 1, [85].log_data[124].valid := 1, [85].time.Year := 2023, [85].time.Month := 1, [85].time.Day := 16, [85].time.Hour := 16, [85].time.Minute := 59, [85].time.Second := 59, [86].log_data[0].min := 1.0, [86].log_data[0].max := 1.0, [86].log_data[0].total := 3600.0, [86].log_data[0].time := 3600.0, [86].log_data[0].valid := 1, [86].log_data[1].time := 3600.0, [86].log_data[1].valid := 1, [86].log_data[2].time := 3600.0, [86].log_data[2].valid := 1, [86].log_data[3].time := 3600.0, [86].log_data[3].valid := 1, [86].log_data[4].time := 3600.0, [86].log_data[4].valid := 1, [86].log_data[5].time := 3600.0, [86].log_data[5].valid := 1, [86].log_data[6].time := 3600.0, [86].log_data[6].valid := 1, [86].log_data[7].time := 3600.0, [86].log_data[7].valid := 1, [86].log_data[8].min := 1.0, [86].log_data[8].max := 1.0, [86].log_data[8].total := 3600.0, [86].log_data[8].time := 3600.0, [86].log_data[8].valid := 1, [86].log_data[9].min := 1.0, [86].log_data[9].max := 1.0, [86].log_data[9].total := 3600.0, [86].log_data[9].time := 3600.0, [86].log_data[9].valid := 1, [86].log_data[10].min := 1.0, [86].log_data[10].max := 1.0, [86].log_data[10].total := 3600.0, [86].log_data[10].time := 3600.0, [86].log_data[10].valid := 1, [86].log_data[11].time := 3600.0, [86].log_data[11].valid := 1, [86].log_data[12].min := 1.0, [86].log_data[12].max := 1.0, [86].log_data[12].total := 3600.0, [86].log_data[12].time := 3600.0, [86].log_data[12].valid := 1, [86].log_data[13].min := 1.0, [86].log_data[13].max := 1.0, [86].log_data[13].total := 3600.0, [86].log_data[13].time := 3600.0, [86].log_data[13].valid := 1, [86].log_data[14].time := 3600.0, [86].log_data[14].valid := 1, [86].log_data[15].time := 3600.0, [86].log_data[15].valid := 1, [86].log_data[16].time := 3600.0, [86].log_data[16].valid := 1,
        [86].log_data[17].min := 1.0, [86].log_data[17].max := 1.0, [86].log_data[17].total := 3600.0, [86].log_data[17].time := 3600.0, [86].log_data[17].valid := 1, [86].log_data[18].time := 3600.0, [86].log_data[18].valid := 1, [86].log_data[19].time := 3600.0, [86].log_data[19].valid := 1, [86].log_data[20].time := 3600.0, [86].log_data[20].valid := 1, [86].log_data[21].min := 1.0, [86].log_data[21].max := 1.0, [86].log_data[21].total := 3600.0, [86].log_data[21].time := 3600.0, [86].log_data[21].valid := 1, [86].log_data[22].time := 3600.0, [86].log_data[22].valid := 1, [86].log_data[23].time := 3600.0, [86].log_data[23].valid := 1, [86].log_data[24].time := 3600.0, [86].log_data[24].valid := 1, [86].log_data[25].time := 3600.0, [86].log_data[25].valid := 1, [86].log_data[26].time := 3600.0, [86].log_data[26].valid := 1, [86].log_data[27].time := 3600.0, [86].log_data[27].valid := 1, [86].log_data[28].time := 3600.0, [86].log_data[28].valid := 1, [86].log_data[29].min := 1.0, [86].log_data[29].max := 1.0, [86].log_data[29].total := 3600.0, [86].log_data[29].time := 3600.0, [86].log_data[29].valid := 1, [86].log_data[30].min := 1.0, [86].log_data[30].max := 1.0, [86].log_data[30].total := 3600.0, [86].log_data[30].time := 3600.0, [86].log_data[30].valid := 1, [86].log_data[31].max := 1.0, [86].log_data[31].total := 1629.7471, [86].log_data[31].time := 3600.0, [86].log_data[31].maxminute := 8, [86].log_data[31].valid := 1, [86].log_data[32].max := 1.0, [86].log_data[32].total := 1520.749, [86].log_data[32].time := 3600.0, [86].log_data[32].minminute := 7, [86].log_data[32].valid := 1, [86].log_data[33].time := 3600.0, [86].log_data[33].valid := 1, [86].log_data[34].time := 3600.0, [86].log_data[34].valid := 1, [86].log_data[35].max := 1.0, [86].log_data[35].total := 1629.7471, [86].log_data[35].time := 3600.0, [86].log_data[35].maxminute := 2, [86].log_data[35].valid := 1, [86].log_data[36].max := 1.0,
        [86].log_data[36].total := 1440.498, [86].log_data[36].time := 3600.0, [86].log_data[36].valid := 1, [86].log_data[37].time := 3600.0, [86].log_data[37].valid := 1, [86].log_data[38].time := 3600.0, [86].log_data[38].valid := 1, [86].log_data[39].min := 0.9934107, [86].log_data[39].max := 1.0044814, [86].log_data[39].total := 3599.212, [86].log_data[39].time := 3600.0, [86].log_data[39].minminute := 44, [86].log_data[39].maxminute := 47, [86].log_data[39].valid := 1, [86].log_data[40].min := 7.5871253, [86].log_data[40].max := 7.603339, [86].log_data[40].total := 27345.953, [86].log_data[40].time := 3600.0, [86].log_data[40].minminute := 21, [86].log_data[40].maxminute := 28, [86].log_data[40].valid := 1, [86].log_data[41].min := 0.022540038, [86].log_data[41].max := 0.028232668, [86].log_data[41].total := 83.212074, [86].log_data[41].time := 3600.0, [86].log_data[41].minminute := 17, [86].log_data[41].maxminute := 1, [86].log_data[41].valid := 1, [86].log_data[42].min := 2.2916427, [86].log_data[42].max := 2.2963536, [86].log_data[42].total := 8259.18, [86].log_data[42].time := 3600.0, [86].log_data[42].minminute := 11, [86].log_data[42].maxminute := 48, [86].log_data[42].valid := 1, [86].log_data[43].min := -0.27999878, [86].log_data[43].max := -0.23999786, [86].log_data[43].total := -936.1721, [86].log_data[43].time := 3600.0, [86].log_data[43].minminute := 51, [86].log_data[43].maxminute := 4, [86].log_data[43].valid := 1, [86].log_data[44].min := -0.30000305, [86].log_data[44].max := -0.27999878, [86].log_data[44].total := -1055.3217, [86].log_data[44].time := 3600.0, [86].log_data[44].valid := 1, [86].log_data[45].time := 3600.0, [86].log_data[45].valid := 1, [86].log_data[46].time := 3600.0, [86].log_data[46].valid := 1, [86].log_data[47].time := 3600.0, [86].log_data[47].valid := 1, [86].log_data[48].min := 6.5708866, [86].log_data[48].max := 6.793755, [86].log_data[48].total := 24135.188, [86].log_data[48].time := 3600.0, [86].log_data[48].minminute := 15, [86].log_data[48].maxminute := 32, [86].log_data[48].valid := 1,
        [86].log_data[49].min := 6.9543743, [86].log_data[49].max := 9.520294, [86].log_data[49].total := 29483.703, [86].log_data[49].time := 3600.0, [86].log_data[49].minminute := 17, [86].log_data[49].maxminute := 59, [86].log_data[49].valid := 1, [86].log_data[50].min := 2.0275915, [86].log_data[50].max := 2.110623, [86].log_data[50].total := 7459.8594, [86].log_data[50].time := 3600.0, [86].log_data[50].minminute := 59, [86].log_data[50].maxminute := 2, [86].log_data[50].valid := 1, [86].log_data[51].time := 3600.0, [86].log_data[51].valid := 1, [86].log_data[52].min := -2.8199997, [86].log_data[52].max := 0.11999512, [86].log_data[52].total := -7758.2393, [86].log_data[52].time := 3600.0, [86].log_data[52].minminute := 50, [86].log_data[52].maxminute := 7, [86].log_data[52].valid := 1, [86].log_data[53].min := -2.4200058, [86].log_data[53].max := 0.2599945, [86].log_data[53].total := -6755.6313, [86].log_data[53].time := 3600.0, [86].log_data[53].minminute := 25, [86].log_data[53].maxminute := 2, [86].log_data[53].valid := 1, [86].log_data[54].max := 0.5325, [86].log_data[54].total := 1251.4119, [86].log_data[54].time := 3600.0, [86].log_data[54].minminute := 7, [86].log_data[54].maxminute := 29, [86].log_data[54].valid := 1, [86].log_data[55].max := 0.50949997, [86].log_data[55].total := 1216.8344, [86].log_data[55].time := 3600.0, [86].log_data[55].maxminute := 2, [86].log_data[55].valid := 1, [86].log_data[56].min := 0.15961748, [86].log_data[56].max := 0.16004932, [86].log_data[56].total := 575.2599, [86].log_data[56].time := 3600.0, [86].log_data[56].minminute := 23, [86].log_data[56].maxminute := 43, [86].log_data[56].valid := 1, [86].log_data[57].min := 0.24641752, [86].log_data[57].max := 0.24885157, [86].log_data[57].total := 890.0368, [86].log_data[57].time := 3600.0, [86].log_data[57].minminute := 53, [86].log_data[57].maxminute := 1, [86].log_data[57].valid := 1, [86].log_data[58].time := 3600.0, [86].log_data[58].valid := 1, [86].log_data[59].time := 3600.0, [86].log_data[59].valid := 1, [86].log_data[60].valid := 1,
        [86].log_data[61].valid := 1, [86].log_data[62].valid := 1, [86].log_data[63].valid := 1, [86].log_data[64].valid := 1, [86].log_data[65].valid := 1, [86].log_data[66].valid := 1, [86].log_data[67].valid := 1, [86].log_data[68].valid := 1, [86].log_data[69].valid := 1, [86].log_data[70].valid := 1, [86].log_data[71].valid := 1, [86].log_data[72].valid := 1, [86].log_data[73].valid := 1, [86].log_data[74].valid := 1, [86].log_data[75].valid := 1, [86].log_data[76].valid := 1, [86].log_data[77].valid := 1, [86].log_data[78].valid := 1, [86].log_data[79].valid := 1, [86].log_data[80].valid := 1, [86].log_data[81].valid := 1, [86].log_data[82].valid := 1, [86].log_data[83].valid := 1, [86].log_data[84].valid := 1, [86].log_data[85].valid := 1, [86].log_data[86].valid := 1, [86].log_data[87].valid := 1, [86].log_data[88].valid := 1, [86].log_data[89].valid := 1, [86].log_data[90].valid := 1, [86].log_data[91].valid := 1, [86].log_data[92].valid := 1, [86].log_data[93].valid := 1, [86].log_data[94].valid := 1, [86].log_data[95].valid := 1, [86].log_data[96].valid := 1, [86].log_data[97].valid := 1, [86].log_data[98].valid := 1, [86].log_data[99].valid := 1, [86].log_data[100].valid := 1, [86].log_data[101].valid := 1, [86].log_data[102].valid := 1, [86].log_data[103].valid := 1, [86].log_data[104].valid := 1, [86].log_data[105].valid := 1, [86].log_data[106].valid := 1, [86].log_data[107].valid := 1, [86].log_data[108].valid := 1, [86].log_data[109].valid := 1, [86].log_data[110].valid := 1, [86].log_data[111].valid := 1, [86].log_data[112].valid := 1, [86].log_data[113].valid := 1, [86].log_data[114].valid := 1, [86].log_data[115].valid := 1, [86].log_data[116].valid := 1, [86].log_data[117].valid := 1, [86].log_data[118].valid := 1, [86].log_data[119].valid := 1, [86].log_data[120].valid := 1,
        [86].log_data[121].valid := 1, [86].log_data[122].valid := 1, [86].log_data[123].valid := 1, [86].log_data[124].valid := 1, [86].time.Year := 2023, [86].time.Month := 1, [86].time.Day := 16, [86].time.Hour := 17, [86].time.Minute := 59, [86].time.Second := 59, [87].log_data[0].min := 1.0, [87].log_data[0].max := 1.0, [87].log_data[0].total := 3600.0, [87].log_data[0].time := 3600.0, [87].log_data[0].valid := 1, [87].log_data[1].max := 1.0, [87].log_data[1].total := 552.5, [87].log_data[1].time := 3600.0, [87].log_data[1].maxminute := 27, [87].log_data[1].valid := 1, [87].log_data[2].max := 1.0, [87].log_data[2].total := 549.0, [87].log_data[2].time := 3600.0, [87].log_data[2].maxminute := 27, [87].log_data[2].valid := 1, [87].log_data[3].time := 3600.0, [87].log_data[3].valid := 1, [87].log_data[4].time := 3600.0, [87].log_data[4].valid := 1, [87].log_data[5].max := 1.0, [87].log_data[5].total := 234.0, [87].log_data[5].time := 3600.0, [87].log_data[5].maxminute := 30, [87].log_data[5].valid := 1, [87].log_data[6].time := 3600.0, [87].log_data[6].valid := 1, [87].log_data[7].time := 3600.0, [87].log_data[7].valid := 1, [87].log_data[8].max := 1.0, [87].log_data[8].total := 2382.0, [87].log_data[8].time := 3600.0, [87].log_data[8].minminute := 11, [87].log_data[8].valid := 1, [87].log_data[9].max := 1.0, [87].log_data[9].total := 2378.5, [87].log_data[9].time := 3600.0, [87].log_data[9].minminute := 11, [87].log_data[9].valid := 1, [87].log_data[10].min := 1.0, [87].log_data[10].max := 1.0, [87].log_data[10].total := 3600.0, [87].log_data[10].time := 3600.0, [87].log_data[10].valid := 1, [87].log_data[11].time := 3600.0, [87].log_data[11].valid := 1, [87].log_data[12].min := 1.0, [87].log_data[12].max := 1.0, [87].log_data[12].total := 3600.0, [87].log_data[12].time := 3600.0, [87].log_data[12].valid := 1,
        [87].log_data[13].min := 1.0, [87].log_data[13].max := 1.0, [87].log_data[13].total := 3600.0, [87].log_data[13].time := 3600.0, [87].log_data[13].valid := 1, [87].log_data[14].time := 3600.0, [87].log_data[14].valid := 1, [87].log_data[15].time := 3600.0, [87].log_data[15].valid := 1, [87].log_data[16].time := 3600.0, [87].log_data[16].valid := 1, [87].log_data[17].min := 1.0, [87].log_data[17].max := 1.0, [87].log_data[17].total := 3600.0, [87].log_data[17].time := 3600.0, [87].log_data[17].valid := 1, [87].log_data[18].time := 3600.0, [87].log_data[18].valid := 1, [87].log_data[19].time := 3600.0, [87].log_data[19].valid := 1, [87].log_data[20].time := 3600.0, [87].log_data[20].valid := 1, [87].log_data[21].min := 1.0, [87].log_data[21].max := 1.0, [87].log_data[21].total := 3600.0, [87].log_data[21].time := 3600.0, [87].log_data[21].valid := 1, [87].log_data[22].time := 3600.0, [87].log_data[22].valid := 1, [87].log_data[23].time := 3600.0, [87].log_data[23].valid := 1, [87].log_data[24].time := 3600.0, [87].log_data[24].valid := 1, [87].log_data[25].time := 3600.0, [87].log_data[25].valid := 1, [87].log_data[26].time := 3600.0, [87].log_data[26].valid := 1, [87].log_data[27].time := 3600.0, [87].log_data[27].valid := 1, [87].log_data[28].time := 3600.0, [87].log_data[28].valid := 1, [87].log_data[29].min := 1.0, [87].log_data[29].max := 1.0, [87].log_data[29].total := 3600.0, [87].log_data[29].time := 3600.0, [87].log_data[29].valid := 1, [87].log_data[30].min := 1.0, [87].log_data[30].max := 1.0, [87].log_data[30].total := 3600.0, [87].log_data[30].time := 3600.0, [87].log_data[30].valid := 1, [87].log_data[31].max := 1.0, [87].log_data[31].total := 958.49805, [87].log_data[31].time := 3600.0, [87].log_data[31].maxminute := 32, [87].log_data[31].valid := 1, [87].log_data[32].max := 1.0, [87].log_data[32].total := 1086.498, [87].log_data[32].time := 3600.0, [87].log_data[32].maxminute := 1,
        [87].log_data[32].valid := 1, [87].log_data[33].time := 3600.0, [87].log_data[33].valid := 1, [87].log_data[34].time := 3600.0, [87].log_data[34].valid := 1, [87].log_data[35].max := 1.0, [87].log_data[35].total := 1079.247, [87].log_data[35].time := 3600.0, [87].log_data[35].maxminute := 5, [87].log_data[35].valid := 1, [87].log_data[36].max := 1.0, [87].log_data[36].total := 942.998, [87].log_data[36].time := 3600.0, [87].log_data[36].minminute := 3, [87].log_data[36].valid := 1, [87].log_data[37].max := 7.3322015, [87].log_data[37].total := 3522.156, [87].log_data[37].time := 3600.0, [87].log_data[37].maxminute := 29, [87].log_data[37].valid := 1, [87].log_data[38].time := 3600.0, [87].log_data[38].valid := 1, [87].log_data[39].min := 0.99376404, [87].log_data[39].max := 1.0212055, [87].log_data[39].total := 3605.9026, [87].log_data[39].time := 3600.0, [87].log_data[39].minminute := 3, [87].log_data[39].maxminute := 30, [87].log_data[39].valid := 1, [87].log_data[40].min := 7.583004, [87].log_data[40].max := 7.6019654, [87].log_data[40].total := 27342.646, [87].log_data[40].time := 3600.0, [87].log_data[40].minminute := 41, [87].log_data[40].maxminute := 50, [87].log_data[40].valid := 1, [87].log_data[41].min := 0.02273633, [87].log_data[41].max := 0.027054932, [87].log_data[41].total := 83.93589, [87].log_data[41].time := 3600.0, [87].log_data[41].maxminute := 10, [87].log_data[41].valid := 1, [87].log_data[42].min := 2.2918782, [87].log_data[42].max := 2.296118, [87].log_data[42].total := 8259.253, [87].log_data[42].time := 3600.0, [87].log_data[42].minminute := 26, [87].log_data[42].maxminute := 9, [87].log_data[42].valid := 1, [87].log_data[43].min := -0.27999878, [87].log_data[43].max := -0.26000214, [87].log_data[43].total := -975.6504, [87].log_data[43].time := 3600.0, [87].log_data[43].valid := 1, [87].log_data[44].min := -0.3199997, [87].log_data[44].max := -0.30000305, [87].log_data[44].total := -1080.1111, [87].log_data[44].time := 3600.0, [87].log_data[44].minminute := 29, [87].log_data[44].valid := 1,
        [87].log_data[45].time := 3600.0, [87].log_data[45].valid := 1, [87].log_data[46].time := 3600.0, [87].log_data[46].valid := 1, [87].log_data[47].time := 3600.0, [87].log_data[47].valid := 1, [87].log_data[48].min := 6.5794053, [87].log_data[48].max := 6.9251137, [87].log_data[48].total := 24220.344, [87].log_data[48].time := 3600.0, [87].log_data[48].minminute := 59, [87].log_data[48].maxminute := 37, [87].log_data[48].valid := 1, [87].log_data[49].min := 6.925912, [87].log_data[49].max := 9.6221695, [87].log_data[49].total := 31373.703, [87].log_data[49].time := 3600.0, [87].log_data[49].minminute := 57, [87].log_data[49].maxminute := 28, [87].log_data[49].valid := 1, [87].log_data[50].min := 1.9989722, [87].log_data[50].max := 2.1512551, [87].log_data[50].total := 7521.0693, [87].log_data[50].time := 3600.0, [87].log_data[50].minminute := 11, [87].log_data[50].maxminute := 31, [87].log_data[50].valid := 1, [87].log_data[51].time := 3600.0, [87].log_data[51].valid := 1, [87].log_data[52].min := -4.3399963, [87].log_data[52].max := 0.11999512, [87].log_data[52].total := -6704.579, [87].log_data[52].time := 3600.0, [87].log_data[52].minminute := 32, [87].log_data[52].valid := 1, [87].log_data[53].min := -4.040001, [87].log_data[53].max := 0.30000305, [87].log_data[53].total := -6065.7534, [87].log_data[53].time := 3600.0, [87].log_data[53].minminute := 32, [87].log_data[53].maxminute := 5, [87].log_data[53].valid := 1, [87].log_data[54].max := 0.5205, [87].log_data[54].total := 810.4983, [87].log_data[54].time := 3600.0, [87].log_data[54].maxminute := 42, [87].log_data[54].valid := 1, [87].log_data[55].max := 0.532, [87].log_data[55].total := 799.77924, [87].log_data[55].time := 3600.0, [87].log_data[55].minminute := 3, [87].log_data[55].maxminute := 57, [87].log_data[55].valid := 1, [87].log_data[56].min := 0.15961748, [87].log_data[56].max := 0.16012783, [87].log_data[56].total := 575.34576, [87].log_data[56].time := 3600.0, [87].log_data[56].minminute := 4, [87].log_data[56].maxminute := 24, [87].log_data[56].valid := 1,
        [87].log_data[57].min := 0.24578941, [87].log_data[57].max := 0.2467316, [87].log_data[57].total := 887.2178, [87].log_data[57].time := 3600.0, [87].log_data[57].minminute := 59, [87].log_data[57].valid := 1, [87].log_data[58].time := 3600.0, [87].log_data[58].valid := 1, [87].log_data[59].time := 3600.0, [87].log_data[59].valid := 1, [87].log_data[60].valid := 1, [87].log_data[61].valid := 1, [87].log_data[62].valid := 1, [87].log_data[63].valid := 1, [87].log_data[64].valid := 1, [87].log_data[65].valid := 1, [87].log_data[66].valid := 1, [87].log_data[67].valid := 1, [87].log_data[68].valid := 1, [87].log_data[69].valid := 1, [87].log_data[70].valid := 1, [87].log_data[71].valid := 1, [87].log_data[72].valid := 1, [87].log_data[73].valid := 1, [87].log_data[74].valid := 1, [87].log_data[75].valid := 1, [87].log_data[76].valid := 1, [87].log_data[77].valid := 1, [87].log_data[78].valid := 1, [87].log_data[79].valid := 1, [87].log_data[80].valid := 1, [87].log_data[81].valid := 1, [87].log_data[82].valid := 1, [87].log_data[83].valid := 1, [87].log_data[84].valid := 1, [87].log_data[85].valid := 1, [87].log_data[86].valid := 1, [87].log_data[87].valid := 1, [87].log_data[88].valid := 1, [87].log_data[89].valid := 1, [87].log_data[90].valid := 1, [87].log_data[91].valid := 1, [87].log_data[92].valid := 1, [87].log_data[93].valid := 1, [87].log_data[94].valid := 1, [87].log_data[95].valid := 1, [87].log_data[96].valid := 1, [87].log_data[97].valid := 1, [87].log_data[98].valid := 1, [87].log_data[99].valid := 1, [87].log_data[100].valid := 1, [87].log_data[101].valid := 1, [87].log_data[102].valid := 1, [87].log_data[103].valid := 1, [87].log_data[104].valid := 1, [87].log_data[105].valid := 1, [87].log_data[106].valid := 1, [87].log_data[107].valid := 1, [87].log_data[108].valid := 1, [87].log_data[109].valid := 1,
        [87].log_data[110].valid := 1, [87].log_data[111].valid := 1, [87].log_data[112].valid := 1, [87].log_data[113].valid := 1, [87].log_data[114].valid := 1, [87].log_data[115].valid := 1, [87].log_data[116].valid := 1, [87].log_data[117].valid := 1, [87].log_data[118].valid := 1, [87].log_data[119].valid := 1, [87].log_data[120].valid := 1, [87].log_data[121].valid := 1, [87].log_data[122].valid := 1, [87].log_data[123].valid := 1, [87].log_data[124].valid := 1, [87].time.Year := 2023, [87].time.Month := 1, [87].time.Day := 16, [87].time.Hour := 18, [87].time.Minute := 59, [87].time.Second := 59, [88].log_data[0].min := 1.0, [88].log_data[0].max := 1.0, [88].log_data[0].total := 3600.0, [88].log_data[0].time := 3600.0, [88].log_data[0].valid := 1, [88].log_data[1].max := 1.0, [88].log_data[1].total := 245.249, [88].log_data[1].time := 3600.0, [88].log_data[1].maxminute := 55, [88].log_data[1].valid := 1, [88].log_data[2].max := 1.0, [88].log_data[2].total := 241.749, [88].log_data[2].time := 3600.0, [88].log_data[2].maxminute := 55, [88].log_data[2].valid := 1, [88].log_data[3].time := 3600.0, [88].log_data[3].valid := 1, [88].log_data[4].time := 3600.0, [88].log_data[4].valid := 1, [88].log_data[5].max := 1.0, [88].log_data[5].total := 96.249, [88].log_data[5].time := 3600.0, [88].log_data[5].maxminute := 58, [88].log_data[5].valid := 1, [88].log_data[6].time := 3600.0, [88].log_data[6].valid := 1, [88].log_data[7].time := 3600.0, [88].log_data[7].valid := 1, [88].log_data[8].min := 1.0, [88].log_data[8].max := 1.0, [88].log_data[8].total := 3600.0, [88].log_data[8].time := 3600.0, [88].log_data[8].valid := 1, [88].log_data[9].min := 1.0, [88].log_data[9].max := 1.0, [88].log_data[9].total := 3600.0, [88].log_data[9].time := 3600.0, [88].log_data[9].valid := 1, [88].log_data[10].min := 1.0,
        [88].log_data[10].max := 1.0, [88].log_data[10].total := 3600.0, [88].log_data[10].time := 3600.0, [88].log_data[10].valid := 1, [88].log_data[11].time := 3600.0, [88].log_data[11].valid := 1, [88].log_data[12].min := 1.0, [88].log_data[12].max := 1.0, [88].log_data[12].total := 3600.0, [88].log_data[12].time := 3600.0, [88].log_data[12].valid := 1, [88].log_data[13].min := 1.0, [88].log_data[13].max := 1.0, [88].log_data[13].total := 3600.0, [88].log_data[13].time := 3600.0, [88].log_data[13].valid := 1, [88].log_data[14].time := 3600.0, [88].log_data[14].valid := 1, [88].log_data[15].time := 3600.0, [88].log_data[15].valid := 1, [88].log_data[16].time := 3600.0, [88].log_data[16].valid := 1, [88].log_data[17].min := 1.0, [88].log_data[17].max := 1.0, [88].log_data[17].total := 3600.0, [88].log_data[17].time := 3600.0, [88].log_data[17].valid := 1, [88].log_data[18].time := 3600.0, [88].log_data[18].valid := 1, [88].log_data[19].time := 3600.0, [88].log_data[19].valid := 1, [88].log_data[20].time := 3600.0, [88].log_data[20].valid := 1, [88].log_data[21].min := 1.0, [88].log_data[21].max := 1.0, [88].log_data[21].total := 3600.0, [88].log_data[21].time := 3600.0, [88].log_data[21].valid := 1, [88].log_data[22].time := 3600.0, [88].log_data[22].valid := 1, [88].log_data[23].time := 3600.0, [88].log_data[23].valid := 1, [88].log_data[24].time := 3600.0, [88].log_data[24].valid := 1, [88].log_data[25].time := 3600.0, [88].log_data[25].valid := 1, [88].log_data[26].time := 3600.0, [88].log_data[26].valid := 1, [88].log_data[27].time := 3600.0, [88].log_data[27].valid := 1, [88].log_data[28].time := 3600.0, [88].log_data[28].valid := 1, [88].log_data[29].min := 1.0, [88].log_data[29].max := 1.0, [88].log_data[29].total := 3600.0, [88].log_data[29].time := 3600.0, [88].log_data[29].valid := 1, [88].log_data[30].min := 1.0, [88].log_data[30].max := 1.0, [88].log_data[30].total := 3600.0,
        [88].log_data[30].time := 3600.0, [88].log_data[30].valid := 1, [88].log_data[31].max := 1.0, [88].log_data[31].total := 1440.7471, [88].log_data[31].time := 3600.0, [88].log_data[31].minminute := 2, [88].log_data[31].valid := 1, [88].log_data[32].max := 1.0, [88].log_data[32].total := 1629.7471, [88].log_data[32].time := 3600.0, [88].log_data[32].maxminute := 3, [88].log_data[32].valid := 1, [88].log_data[33].time := 3600.0, [88].log_data[33].valid := 1, [88].log_data[34].time := 3600.0, [88].log_data[34].valid := 1, [88].log_data[35].max := 1.0, [88].log_data[35].total := 1471.249, [88].log_data[35].time := 3600.0, [88].log_data[35].minminute := 6, [88].log_data[35].valid := 1, [88].log_data[36].max := 1.0, [88].log_data[36].total := 1629.7471, [88].log_data[36].time := 3600.0, [88].log_data[36].maxminute := 7, [88].log_data[36].valid := 1, [88].log_data[37].max := 7.469998, [88].log_data[37].total := 1804.7146, [88].log_data[37].time := 3600.0, [88].log_data[37].maxminute := 56, [88].log_data[37].valid := 1, [88].log_data[38].time := 3600.0, [88].log_data[38].valid := 1, [88].log_data[39].min := 0.9956484, [88].log_data[39].max := 1.0216767, [88].log_data[39].total := 3606.4849, [88].log_data[39].time := 3600.0, [88].log_data[39].minminute := 24, [88].log_data[39].maxminute := 58, [88].log_data[39].valid := 1, [88].log_data[40].min := 7.5827284, [88].log_data[40].max := 7.604989, [88].log_data[40].total := 27346.25, [88].log_data[40].time := 3600.0, [88].log_data[40].minminute := 3, [88].log_data[40].maxminute := 57, [88].log_data[40].valid := 1, [88].log_data[41].min := 0.02273633, [88].log_data[41].max := 0.03333618, [88].log_data[41].total := 88.96635, [88].log_data[41].time := 3600.0, [88].log_data[41].maxminute := 28, [88].log_data[41].valid := 1, [88].log_data[42].min := 2.2918782, [88].log_data[42].max := 2.2963536, [88].log_data[42].total := 8259.308, [88].log_data[42].time := 3600.0, [88].log_data[42].minminute := 3, [88].log_data[42].maxminute := 44, [88].log_data[42].valid := 1,
        [88].log_data[43].min := -0.27999878, [88].log_data[43].max := -0.26000214, [88].log_data[43].total := -1006.83765, [88].log_data[43].time := 3600.0, [88].log_data[43].valid := 1, [88].log_data[44].min := -0.3199997, [88].log_data[44].max := -0.30000305, [88].log_data[44].total := -1080.7336, [88].log_data[44].time := 3600.0, [88].log_data[44].minminute := 5, [88].log_data[44].valid := 1, [88].log_data[45].time := 3600.0, [88].log_data[45].valid := 1, [88].log_data[46].time := 3600.0, [88].log_data[46].valid := 1, [88].log_data[47].time := 3600.0, [88].log_data[47].valid := 1, [88].log_data[48].min := 6.578306, [88].log_data[48].max := 6.85806, [88].log_data[48].total := 24284.729, [88].log_data[48].time := 3600.0, [88].log_data[48].minminute := 1, [88].log_data[48].maxminute := 59, [88].log_data[48].valid := 1, [88].log_data[49].min := 7.1131735, [88].log_data[49].max := 9.591745, [88].log_data[49].total := 32329.21, [88].log_data[49].time := 3600.0, [88].log_data[49].minminute := 2, [88].log_data[49].maxminute := 56, [88].log_data[49].valid := 1, [88].log_data[50].min := 2.0019166, [88].log_data[50].max := 2.0960188, [88].log_data[50].total := 7380.733, [88].log_data[50].time := 3600.0, [88].log_data[50].minminute := 57, [88].log_data[50].valid := 1, [88].log_data[51].time := 3600.0, [88].log_data[51].valid := 1, [88].log_data[52].min := -2.880005, [88].log_data[52].max := 0.11999512, [88].log_data[52].total := -7547.557, [88].log_data[52].time := 3600.0, [88].log_data[52].minminute := 14, [88].log_data[52].maxminute := 2, [88].log_data[52].valid := 1, [88].log_data[53].min := -2.6600037, [88].log_data[53].max := 0.27999878, [88].log_data[53].total := -6900.551, [88].log_data[53].time := 3600.0, [88].log_data[53].minminute := 18, [88].log_data[53].maxminute := 7, [88].log_data[53].valid := 1, [88].log_data[54].max := 0.509, [88].log_data[54].total := 1216.8668, [88].log_data[54].time := 3600.0, [88].log_data[54].minminute := 2, [88].log_data[54].maxminute := 14, [88].log_data[54].valid := 1, [88].log_data[55].max := 0.561,
        [88].log_data[55].total := 1231.4576, [88].log_data[55].time := 3600.0, [88].log_data[55].minminute := 6, [88].log_data[55].maxminute := 18, [88].log_data[55].valid := 1, [88].log_data[56].min := 0.15965673, [88].log_data[56].max := 0.16016708, [88].log_data[56].total := 575.5861, [88].log_data[56].time := 3600.0, [88].log_data[56].minminute := 17, [88].log_data[56].maxminute := 50, [88].log_data[56].valid := 1, [88].log_data[57].min := 0.24417979, [88].log_data[57].max := 0.24598569, [88].log_data[57].total := 880.1043, [88].log_data[57].time := 3600.0, [88].log_data[57].minminute := 51, [88].log_data[57].valid := 1, [88].log_data[58].time := 3600.0, [88].log_data[58].valid := 1, [88].log_data[59].time := 3600.0, [88].log_data[59].valid := 1, [88].log_data[60].valid := 1, [88].log_data[61].valid := 1, [88].log_data[62].valid := 1, [88].log_data[63].valid := 1, [88].log_data[64].valid := 1, [88].log_data[65].valid := 1, [88].log_data[66].valid := 1, [88].log_data[67].valid := 1, [88].log_data[68].valid := 1, [88].log_data[69].valid := 1, [88].log_data[70].valid := 1, [88].log_data[71].valid := 1, [88].log_data[72].valid := 1, [88].log_data[73].valid := 1, [88].log_data[74].valid := 1, [88].log_data[75].valid := 1, [88].log_data[76].valid := 1, [88].log_data[77].valid := 1, [88].log_data[78].valid := 1, [88].log_data[79].valid := 1, [88].log_data[80].valid := 1, [88].log_data[81].valid := 1, [88].log_data[82].valid := 1, [88].log_data[83].valid := 1, [88].log_data[84].valid := 1, [88].log_data[85].valid := 1, [88].log_data[86].valid := 1, [88].log_data[87].valid := 1, [88].log_data[88].valid := 1, [88].log_data[89].valid := 1, [88].log_data[90].valid := 1, [88].log_data[91].valid := 1, [88].log_data[92].valid := 1, [88].log_data[93].valid := 1, [88].log_data[94].valid := 1, [88].log_data[95].valid := 1, [88].log_data[96].valid := 1, [88].log_data[97].valid := 1,
        [88].log_data[98].valid := 1, [88].log_data[99].valid := 1, [88].log_data[100].valid := 1, [88].log_data[101].valid := 1, [88].log_data[102].valid := 1, [88].log_data[103].valid := 1, [88].log_data[104].valid := 1, [88].log_data[105].valid := 1, [88].log_data[106].valid := 1, [88].log_data[107].valid := 1, [88].log_data[108].valid := 1, [88].log_data[109].valid := 1, [88].log_data[110].valid := 1, [88].log_data[111].valid := 1, [88].log_data[112].valid := 1, [88].log_data[113].valid := 1, [88].log_data[114].valid := 1, [88].log_data[115].valid := 1, [88].log_data[116].valid := 1, [88].log_data[117].valid := 1, [88].log_data[118].valid := 1, [88].log_data[119].valid := 1, [88].log_data[120].valid := 1, [88].log_data[121].valid := 1, [88].log_data[122].valid := 1, [88].log_data[123].valid := 1, [88].log_data[124].valid := 1, [88].time.Year := 2023, [88].time.Month := 1, [88].time.Day := 16, [88].time.Hour := 19, [88].time.Minute := 59, [88].time.Second := 59, [89].log_data[0].min := 1.0, [89].log_data[0].max := 1.0, [89].log_data[0].total := 3600.0, [89].log_data[0].time := 3600.0, [89].log_data[0].valid := 1, [89].log_data[1].max := 1.0, [89].log_data[1].total := 305.751, [89].log_data[1].time := 3600.0, [89].log_data[1].minminute := 5, [89].log_data[1].valid := 1, [89].log_data[2].max := 1.0, [89].log_data[2].total := 305.751, [89].log_data[2].time := 3600.0, [89].log_data[2].minminute := 5, [89].log_data[2].valid := 1, [89].log_data[3].time := 3600.0, [89].log_data[3].valid := 1, [89].log_data[4].time := 3600.0, [89].log_data[4].valid := 1, [89].log_data[5].max := 1.0, [89].log_data[5].total := 143.251, [89].log_data[5].time := 3600.0, [89].log_data[5].valid := 1, [89].log_data[6].time := 3600.0, [89].log_data[6].valid := 1, [89].log_data[7].time := 3600.0, [89].log_data[7].valid := 1,
        [89].log_data[8].min := 1.0, [89].log_data[8].max := 1.0, [89].log_data[8].total := 3600.0, [89].log_data[8].time := 3600.0, [89].log_data[8].valid := 1, [89].log_data[9].min := 1.0, [89].log_data[9].max := 1.0, [89].log_data[9].total := 3600.0, [89].log_data[9].time := 3600.0, [89].log_data[9].valid := 1, [89].log_data[10].min := 1.0, [89].log_data[10].max := 1.0, [89].log_data[10].total := 3600.0, [89].log_data[10].time := 3600.0, [89].log_data[10].valid := 1, [89].log_data[11].time := 3600.0, [89].log_data[11].valid := 1, [89].log_data[12].min := 1.0, [89].log_data[12].max := 1.0, [89].log_data[12].total := 3600.0, [89].log_data[12].time := 3600.0, [89].log_data[12].valid := 1, [89].log_data[13].min := 1.0, [89].log_data[13].max := 1.0, [89].log_data[13].total := 3600.0, [89].log_data[13].time := 3600.0, [89].log_data[13].valid := 1, [89].log_data[14].time := 3600.0, [89].log_data[14].valid := 1, [89].log_data[15].time := 3600.0, [89].log_data[15].valid := 1, [89].log_data[16].time := 3600.0, [89].log_data[16].valid := 1, [89].log_data[17].min := 1.0, [89].log_data[17].max := 1.0, [89].log_data[17].total := 3600.0, [89].log_data[17].time := 3600.0, [89].log_data[17].valid := 1, [89].log_data[18].time := 3600.0, [89].log_data[18].valid := 1, [89].log_data[19].time := 3600.0, [89].log_data[19].valid := 1, [89].log_data[20].time := 3600.0, [89].log_data[20].valid := 1, [89].log_data[21].min := 1.0, [89].log_data[21].max := 1.0, [89].log_data[21].total := 3600.0, [89].log_data[21].time := 3600.0, [89].log_data[21].valid := 1, [89].log_data[22].time := 3600.0, [89].log_data[22].valid := 1, [89].log_data[23].time := 3600.0, [89].log_data[23].valid := 1, [89].log_data[24].time := 3600.0, [89].log_data[24].valid := 1, [89].log_data[25].time := 3600.0, [89].log_data[25].valid := 1, [89].log_data[26].time := 3600.0, [89].log_data[26].valid := 1, [89].log_data[27].time := 3600.0,
        [89].log_data[27].valid := 1, [89].log_data[28].time := 3600.0, [89].log_data[28].valid := 1, [89].log_data[29].min := 1.0, [89].log_data[29].max := 1.0, [89].log_data[29].total := 3600.0, [89].log_data[29].time := 3600.0, [89].log_data[29].valid := 1, [89].log_data[30].min := 1.0, [89].log_data[30].max := 1.0, [89].log_data[30].total := 3600.0, [89].log_data[30].time := 3600.0, [89].log_data[30].valid := 1, [89].log_data[31].max := 1.0, [89].log_data[31].total := 1440.7471, [89].log_data[31].time := 3600.0, [89].log_data[31].minminute := 5, [89].log_data[31].valid := 1, [89].log_data[32].max := 1.0, [89].log_data[32].total := 1629.998, [89].log_data[32].time := 3600.0, [89].log_data[32].maxminute := 6, [89].log_data[32].valid := 1, [89].log_data[33].time := 3600.0, [89].log_data[33].valid := 1, [89].log_data[34].time := 3600.0, [89].log_data[34].valid := 1, [89].log_data[35].max := 1.0, [89].log_data[35].total := 1629.7471, [89].log_data[35].time := 3600.0, [89].log_data[35].valid := 1, [89].log_data[36].max := 1.0, [89].log_data[36].total := 1498.2471, [89].log_data[36].time := 3600.0, [89].log_data[36].maxminute := 11, [89].log_data[36].valid := 1, [89].log_data[37].max := 7.3671417, [89].log_data[37].total := 1778.3265, [89].log_data[37].time := 3600.0, [89].log_data[37].minminute := 4, [89].log_data[37].valid := 1, [89].log_data[38].time := 3600.0, [89].log_data[38].valid := 1, [89].log_data[39].min := 0.995884, [89].log_data[39].max := 1.0207345, [89].log_data[39].total := 3608.6467, [89].log_data[39].time := 3600.0, [89].log_data[39].minminute := 50, [89].log_data[39].maxminute := 2, [89].log_data[39].valid := 1, [89].log_data[40].min := 7.577233, [89].log_data[40].max := 7.609111, [89].log_data[40].total := 27342.379, [89].log_data[40].time := 3600.0, [89].log_data[40].minminute := 42, [89].log_data[40].maxminute := 4, [89].log_data[40].valid := 1, [89].log_data[41].min := 0.022540038, [89].log_data[41].max := 0.023128908, [89].log_data[41].total := 82.48046,
        [89].log_data[41].time := 3600.0, [89].log_data[41].minminute := 29, [89].log_data[41].valid := 1, [89].log_data[42].min := 2.2916427, [89].log_data[42].max := 2.296236, [89].log_data[42].total := 8259.296, [89].log_data[42].time := 3600.0, [89].log_data[42].minminute := 35, [89].log_data[42].maxminute := 42, [89].log_data[42].valid := 1, [89].log_data[43].min := -0.27999878, [89].log_data[43].max := -0.26000214, [89].log_data[43].total := -1007.2124, [89].log_data[43].time := 3600.0, [89].log_data[43].valid := 1, [89].log_data[44].min := -0.3199997, [89].log_data[44].max := -0.30000305, [89].log_data[44].total := -1083.9048, [89].log_data[44].time := 3600.0, [89].log_data[44].valid := 1, [89].log_data[45].time := 3600.0, [89].log_data[45].valid := 1, [89].log_data[46].time := 3600.0, [89].log_data[46].valid := 1, [89].log_data[47].time := 3600.0, [89].log_data[47].valid := 1, [89].log_data[48].min := 6.578031, [89].log_data[48].max := 6.939678, [89].log_data[48].total := 24220.031, [89].log_data[48].time := 3600.0, [89].log_data[48].minminute := 26, [89].log_data[48].maxminute := 1, [89].log_data[48].valid := 1, [89].log_data[49].min := 6.8974495, [89].log_data[49].max := 9.402521, [89].log_data[49].total := 29130.998, [89].log_data[49].time := 3600.0, [89].log_data[49].minminute := 27, [89].log_data[49].maxminute := 59, [89].log_data[49].valid := 1, [89].log_data[50].min := 2.042549, [89].log_data[50].max := 2.1139205, [89].log_data[50].total := 7487.696, [89].log_data[50].time := 3600.0, [89].log_data[50].minminute := 59, [89].log_data[50].maxminute := 7, [89].log_data[50].valid := 1, [89].log_data[51].time := 3600.0, [89].log_data[51].valid := 1, [89].log_data[52].min := -3.0, [89].log_data[52].max := 0.11999512, [89].log_data[52].total := -7585.6196, [89].log_data[52].time := 3600.0, [89].log_data[52].minminute := 48, [89].log_data[52].maxminute := 5, [89].log_data[52].valid := 1, [89].log_data[53].min := -2.4400024, [89].log_data[53].max := 0.30000305, [89].log_data[53].total := -7000.086, [89].log_data[53].time := 3600.0,
        [89].log_data[53].minminute := 1, [89].log_data[53].maxminute := 10, [89].log_data[53].valid := 1, [89].log_data[54].max := 0.5385, [89].log_data[54].total := 1217.3622, [89].log_data[54].time := 3600.0, [89].log_data[54].minminute := 5, [89].log_data[54].maxminute := 38, [89].log_data[54].valid := 1, [89].log_data[55].max := 0.5255, [89].log_data[55].total := 1239.965, [89].log_data[55].time := 3600.0, [89].log_data[55].maxminute := 42, [89].log_data[55].valid := 1, [89].log_data[56].min := 0.159696, [89].log_data[56].max := 0.16016708, [89].log_data[56].total := 575.7408, [89].log_data[56].time := 3600.0, [89].log_data[56].minminute := 2, [89].log_data[56].maxminute := 8, [89].log_data[56].valid := 1, [89].log_data[57].min := 0.24225615, [89].log_data[57].max := 0.24457242, [89].log_data[57].total := 876.0598, [89].log_data[57].time := 3600.0, [89].log_data[57].minminute := 36, [89].log_data[57].maxminute := 8, [89].log_data[57].valid := 1, [89].log_data[58].time := 3600.0, [89].log_data[58].valid := 1, [89].log_data[59].time := 3600.0, [89].log_data[59].valid := 1, [89].log_data[60].valid := 1, [89].log_data[61].valid := 1, [89].log_data[62].valid := 1, [89].log_data[63].valid := 1, [89].log_data[64].valid := 1, [89].log_data[65].valid := 1, [89].log_data[66].valid := 1, [89].log_data[67].valid := 1, [89].log_data[68].valid := 1, [89].log_data[69].valid := 1, [89].log_data[70].valid := 1, [89].log_data[71].valid := 1, [89].log_data[72].valid := 1, [89].log_data[73].valid := 1, [89].log_data[74].valid := 1, [89].log_data[75].valid := 1, [89].log_data[76].valid := 1, [89].log_data[77].valid := 1, [89].log_data[78].valid := 1, [89].log_data[79].valid := 1, [89].log_data[80].valid := 1, [89].log_data[81].valid := 1, [89].log_data[82].valid := 1, [89].log_data[83].valid := 1, [89].log_data[84].valid := 1, [89].log_data[85].valid := 1, [89].log_data[86].valid := 1, [89].log_data[87].valid := 1,
        [89].log_data[88].valid := 1, [89].log_data[89].valid := 1, [89].log_data[90].valid := 1, [89].log_data[91].valid := 1, [89].log_data[92].valid := 1, [89].log_data[93].valid := 1, [89].log_data[94].valid := 1, [89].log_data[95].valid := 1, [89].log_data[96].valid := 1, [89].log_data[97].valid := 1, [89].log_data[98].valid := 1, [89].log_data[99].valid := 1, [89].log_data[100].valid := 1, [89].log_data[101].valid := 1, [89].log_data[102].valid := 1, [89].log_data[103].valid := 1, [89].log_data[104].valid := 1, [89].log_data[105].valid := 1, [89].log_data[106].valid := 1, [89].log_data[107].valid := 1, [89].log_data[108].valid := 1, [89].log_data[109].valid := 1, [89].log_data[110].valid := 1, [89].log_data[111].valid := 1, [89].log_data[112].valid := 1, [89].log_data[113].valid := 1, [89].log_data[114].valid := 1, [89].log_data[115].valid := 1, [89].log_data[116].valid := 1, [89].log_data[117].valid := 1, [89].log_data[118].valid := 1, [89].log_data[119].valid := 1, [89].log_data[120].valid := 1, [89].log_data[121].valid := 1, [89].log_data[122].valid := 1, [89].log_data[123].valid := 1, [89].log_data[124].valid := 1, [89].time.Year := 2023, [89].time.Month := 1, [89].time.Day := 16, [89].time.Hour := 20, [89].time.Minute := 59, [89].time.Second := 59, [90].log_data[0].min := 1.0, [90].log_data[0].max := 1.0, [90].log_data[0].total := 3599.5, [90].log_data[0].time := 3599.5, [90].log_data[0].valid := 1, [90].log_data[1].max := 1.0, [90].log_data[1].total := 575.5, [90].log_data[1].time := 3599.5, [90].log_data[1].maxminute := 4, [90].log_data[1].valid := 1, [90].log_data[2].max := 1.0, [90].log_data[2].total := 572.0, [90].log_data[2].time := 3599.5, [90].log_data[2].maxminute := 4, [90].log_data[2].valid := 1, [90].log_data[3].time := 3599.5, [90].log_data[3].valid := 1,
        [90].log_data[4].time := 3599.5, [90].log_data[4].valid := 1, [90].log_data[5].max := 1.0, [90].log_data[5].total := 245.5, [90].log_data[5].time := 3599.5, [90].log_data[5].maxminute := 6, [90].log_data[5].valid := 1, [90].log_data[6].time := 3599.5, [90].log_data[6].valid := 1, [90].log_data[7].time := 3599.5, [90].log_data[7].valid := 1, [90].log_data[8].min := 1.0, [90].log_data[8].max := 1.0, [90].log_data[8].total := 3599.5, [90].log_data[8].time := 3599.5, [90].log_data[8].valid := 1, [90].log_data[9].min := 1.0, [90].log_data[9].max := 1.0, [90].log_data[9].total := 3599.5, [90].log_data[9].time := 3599.5, [90].log_data[9].valid := 1, [90].log_data[10].min := 1.0, [90].log_data[10].max := 1.0, [90].log_data[10].total := 3599.5, [90].log_data[10].time := 3599.5, [90].log_data[10].valid := 1, [90].log_data[11].time := 3599.5, [90].log_data[11].valid := 1, [90].log_data[12].min := 1.0, [90].log_data[12].max := 1.0, [90].log_data[12].total := 3599.5, [90].log_data[12].time := 3599.5, [90].log_data[12].valid := 1, [90].log_data[13].min := 1.0, [90].log_data[13].max := 1.0, [90].log_data[13].total := 3599.5, [90].log_data[13].time := 3599.5, [90].log_data[13].valid := 1, [90].log_data[14].time := 3599.5, [90].log_data[14].valid := 1, [90].log_data[15].time := 3599.5, [90].log_data[15].valid := 1, [90].log_data[16].time := 3599.5, [90].log_data[16].valid := 1, [90].log_data[17].min := 1.0, [90].log_data[17].max := 1.0, [90].log_data[17].total := 3599.5, [90].log_data[17].time := 3599.5, [90].log_data[17].valid := 1, [90].log_data[18].time := 3599.5, [90].log_data[18].valid := 1, [90].log_data[19].time := 3599.5, [90].log_data[19].valid := 1, [90].log_data[20].time := 3599.5, [90].log_data[20].valid := 1, [90].log_data[21].min := 1.0, [90].log_data[21].max := 1.0, [90].log_data[21].total := 3599.5, [90].log_data[21].time := 3599.5, [90].log_data[21].valid := 1,
        [90].log_data[22].time := 3599.5, [90].log_data[22].valid := 1, [90].log_data[23].time := 3599.5, [90].log_data[23].valid := 1, [90].log_data[24].time := 3599.5, [90].log_data[24].valid := 1, [90].log_data[25].time := 3599.5, [90].log_data[25].valid := 1, [90].log_data[26].time := 3599.5, [90].log_data[26].valid := 1, [90].log_data[27].time := 3599.5, [90].log_data[27].valid := 1, [90].log_data[28].time := 3599.5, [90].log_data[28].valid := 1, [90].log_data[29].min := 1.0, [90].log_data[29].max := 1.0, [90].log_data[29].total := 3599.5, [90].log_data[29].time := 3599.5, [90].log_data[29].valid := 1, [90].log_data[30].min := 1.0, [90].log_data[30].max := 1.0, [90].log_data[30].total := 3599.5, [90].log_data[30].time := 3599.5, [90].log_data[30].valid := 1, [90].log_data[31].max := 1.0, [90].log_data[31].total := 1592.498, [90].log_data[31].time := 3599.5, [90].log_data[31].minminute := 8, [90].log_data[31].valid := 1, [90].log_data[32].max := 1.0, [90].log_data[32].total := 1565.998, [90].log_data[32].time := 3599.5, [90].log_data[32].maxminute := 9, [90].log_data[32].valid := 1, [90].log_data[33].time := 3599.5, [90].log_data[33].valid := 1, [90].log_data[34].time := 3599.5, [90].log_data[34].valid := 1, [90].log_data[35].max := 1.0, [90].log_data[35].total := 1629.7471, [90].log_data[35].time := 3599.5, [90].log_data[35].maxminute := 3, [90].log_data[35].valid := 1, [90].log_data[36].max := 1.0, [90].log_data[36].total := 1440.2471, [90].log_data[36].time := 3599.5, [90].log_data[36].minminute := 2, [90].log_data[36].valid := 1, [90].log_data[37].max := 7.2116785, [90].log_data[37].total := 3622.532, [90].log_data[37].time := 3599.5, [90].log_data[37].maxminute := 5, [90].log_data[37].valid := 1, [90].log_data[38].time := 3599.5, [90].log_data[38].valid := 1, [90].log_data[39].min := 0.9960017, [90].log_data[39].max := 1.0222654, [90].log_data[39].total := 3609.743, [90].log_data[39].time := 3599.5, [90].log_data[39].minminute := 27,
        [90].log_data[39].maxminute := 11, [90].log_data[39].valid := 1, [90].log_data[40].min := 7.5816298, [90].log_data[40].max := 7.6077366, [90].log_data[40].total := 27344.992, [90].log_data[40].time := 3599.5, [90].log_data[40].minminute := 2, [90].log_data[40].maxminute := 36, [90].log_data[40].valid := 1, [90].log_data[41].min := 0.02273633, [90].log_data[41].max := 0.023128908, [90].log_data[41].total := 82.47191, [90].log_data[41].time := 3599.5, [90].log_data[41].valid := 1, [90].log_data[42].min := 2.2916427, [90].log_data[42].max := 2.2963536, [90].log_data[42].total := 8258.176, [90].log_data[42].time := 3599.5, [90].log_data[42].minminute := 1, [90].log_data[42].maxminute := 25, [90].log_data[42].valid := 1, [90].log_data[43].min := -0.27999878, [90].log_data[43].max := -0.26000214, [90].log_data[43].total := -1007.10724, [90].log_data[43].time := 3599.5, [90].log_data[43].maxminute := 1, [90].log_data[43].valid := 1, [90].log_data[44].min := -0.3199997, [90].log_data[44].max := -0.30000305, [90].log_data[44].total := -1081.9528, [90].log_data[44].time := 3599.5, [90].log_data[44].valid := 1, [90].log_data[45].time := 3599.5, [90].log_data[45].valid := 1, [90].log_data[46].time := 3599.5, [90].log_data[46].valid := 1, [90].log_data[47].time := 3599.5, [90].log_data[47].valid := 1, [90].log_data[48].min := 6.581329, [90].log_data[48].max := 6.905327, [90].log_data[48].total := 24212.178, [90].log_data[48].time := 3599.5, [90].log_data[48].minminute := 36, [90].log_data[48].maxminute := 9, [90].log_data[48].valid := 1, [90].log_data[49].min := 6.9015718, [90].log_data[49].max := 9.507143, [90].log_data[49].total := 28990.12, [90].log_data[49].time := 3599.5, [90].log_data[49].minminute := 32, [90].log_data[49].maxminute := 7, [90].log_data[49].valid := 1, [90].log_data[50].min := 2.0338335, [90].log_data[50].max := 2.1458375, [90].log_data[50].total := 7578.8013, [90].log_data[50].time := 3599.5, [90].log_data[50].minminute := 6, [90].log_data[50].maxminute := 14, [90].log_data[50].valid := 1, [90].log_data[51].time := 3599.5,
        [90].log_data[51].valid := 1, [90].log_data[52].min := -2.9000015, [90].log_data[52].max := 0.11999512, [90].log_data[52].total := -7815.945, [90].log_data[52].time := 3599.5, [90].log_data[52].minminute := 41, [90].log_data[52].maxminute := 8, [90].log_data[52].valid := 1, [90].log_data[53].min := -2.4800034, [90].log_data[53].max := 0.30000305, [90].log_data[53].total := -6969.5854, [90].log_data[53].time := 3599.5, [90].log_data[53].minminute := 6, [90].log_data[53].maxminute := 3, [90].log_data[53].valid := 1, [90].log_data[54].max := 0.546, [90].log_data[54].total := 1254.1052, [90].log_data[54].time := 3599.5, [90].log_data[54].minminute := 8, [90].log_data[54].maxminute := 10, [90].log_data[54].valid := 1, [90].log_data[55].max := 0.5265, [90].log_data[55].total := 1216.8901, [90].log_data[55].time := 3599.5, [90].log_data[55].minminute := 2, [90].log_data[55].maxminute := 45, [90].log_data[55].valid := 1, [90].log_data[56].min := 0.15981378, [90].log_data[56].max := 0.16020635, [90].log_data[56].total := 575.81494, [90].log_data[56].time := 3599.5, [90].log_data[56].maxminute := 4, [90].log_data[56].valid := 1, [90].log_data[57].min := 0.24048956, [90].log_data[57].max := 0.24260947, [90].log_data[57].total := 870.2085, [90].log_data[57].time := 3599.5, [90].log_data[57].minminute := 45, [90].log_data[57].maxminute := 4, [90].log_data[57].valid := 1, [90].log_data[58].time := 3599.5, [90].log_data[58].valid := 1, [90].log_data[59].time := 3599.5, [90].log_data[59].valid := 1, [90].log_data[60].valid := 1, [90].log_data[61].valid := 1, [90].log_data[62].valid := 1, [90].log_data[63].valid := 1, [90].log_data[64].valid := 1, [90].log_data[65].valid := 1, [90].log_data[66].valid := 1, [90].log_data[67].valid := 1, [90].log_data[68].valid := 1, [90].log_data[69].valid := 1, [90].log_data[70].valid := 1, [90].log_data[71].valid := 1, [90].log_data[72].valid := 1, [90].log_data[73].valid := 1, [90].log_data[74].valid := 1, [90].log_data[75].valid := 1,
        [90].log_data[76].valid := 1, [90].log_data[77].valid := 1, [90].log_data[78].valid := 1, [90].log_data[79].valid := 1, [90].log_data[80].valid := 1, [90].log_data[81].valid := 1, [90].log_data[82].valid := 1, [90].log_data[83].valid := 1, [90].log_data[84].valid := 1, [90].log_data[85].valid := 1, [90].log_data[86].valid := 1, [90].log_data[87].valid := 1, [90].log_data[88].valid := 1, [90].log_data[89].valid := 1, [90].log_data[90].valid := 1, [90].log_data[91].valid := 1, [90].log_data[92].valid := 1, [90].log_data[93].valid := 1, [90].log_data[94].valid := 1, [90].log_data[95].valid := 1, [90].log_data[96].valid := 1, [90].log_data[97].valid := 1, [90].log_data[98].valid := 1, [90].log_data[99].valid := 1, [90].log_data[100].valid := 1, [90].log_data[101].valid := 1, [90].log_data[102].valid := 1, [90].log_data[103].valid := 1, [90].log_data[104].valid := 1, [90].log_data[105].valid := 1, [90].log_data[106].valid := 1, [90].log_data[107].valid := 1, [90].log_data[108].valid := 1, [90].log_data[109].valid := 1, [90].log_data[110].valid := 1, [90].log_data[111].valid := 1, [90].log_data[112].valid := 1, [90].log_data[113].valid := 1, [90].log_data[114].valid := 1, [90].log_data[115].valid := 1, [90].log_data[116].valid := 1, [90].log_data[117].valid := 1, [90].log_data[118].valid := 1, [90].log_data[119].valid := 1, [90].log_data[120].valid := 1, [90].log_data[121].valid := 1, [90].log_data[122].valid := 1, [90].log_data[123].valid := 1, [90].log_data[124].valid := 1, [90].time.Year := 2023, [90].time.Month := 1, [90].time.Day := 16, [90].time.Hour := 21, [90].time.Minute := 59, [90].time.Second := 59, [91].log_data[0].min := 1.0, [91].log_data[0].max := 1.0, [91].log_data[0].total := 3600.0, [91].log_data[0].time := 3600.0, [91].log_data[0].valid := 1,
        [91].log_data[1].max := 1.0, [91].log_data[1].total := 550.0, [91].log_data[1].time := 3600.0, [91].log_data[1].maxminute := 18, [91].log_data[1].valid := 1, [91].log_data[2].max := 1.0, [91].log_data[2].total := 546.5, [91].log_data[2].time := 3600.0, [91].log_data[2].maxminute := 18, [91].log_data[2].valid := 1, [91].log_data[3].time := 3600.0, [91].log_data[3].valid := 1, [91].log_data[4].time := 3600.0, [91].log_data[4].valid := 1, [91].log_data[5].max := 1.0, [91].log_data[5].total := 246.0, [91].log_data[5].time := 3600.0, [91].log_data[5].maxminute := 21, [91].log_data[5].valid := 1, [91].log_data[6].time := 3600.0, [91].log_data[6].valid := 1, [91].log_data[7].time := 3600.0, [91].log_data[7].valid := 1, [91].log_data[8].min := 1.0, [91].log_data[8].max := 1.0, [91].log_data[8].total := 3600.0, [91].log_data[8].time := 3600.0, [91].log_data[8].valid := 1, [91].log_data[9].min := 1.0, [91].log_data[9].max := 1.0, [91].log_data[9].total := 3600.0, [91].log_data[9].time := 3600.0, [91].log_data[9].valid := 1, [91].log_data[10].min := 1.0, [91].log_data[10].max := 1.0, [91].log_data[10].total := 3600.0, [91].log_data[10].time := 3600.0, [91].log_data[10].valid := 1, [91].log_data[11].time := 3600.0, [91].log_data[11].valid := 1, [91].log_data[12].min := 1.0, [91].log_data[12].max := 1.0, [91].log_data[12].total := 3600.0, [91].log_data[12].time := 3600.0, [91].log_data[12].valid := 1, [91].log_data[13].min := 1.0, [91].log_data[13].max := 1.0, [91].log_data[13].total := 3600.0, [91].log_data[13].time := 3600.0, [91].log_data[13].valid := 1, [91].log_data[14].time := 3600.0, [91].log_data[14].valid := 1, [91].log_data[15].time := 3600.0, [91].log_data[15].valid := 1, [91].log_data[16].time := 3600.0, [91].log_data[16].valid := 1, [91].log_data[17].min := 1.0, [91].log_data[17].max := 1.0, [91].log_data[17].total := 3600.0, [91].log_data[17].time := 3600.0,
        [91].log_data[17].valid := 1, [91].log_data[18].time := 3600.0, [91].log_data[18].valid := 1, [91].log_data[19].time := 3600.0, [91].log_data[19].valid := 1, [91].log_data[20].time := 3600.0, [91].log_data[20].valid := 1, [91].log_data[21].min := 1.0, [91].log_data[21].max := 1.0, [91].log_data[21].total := 3600.0, [91].log_data[21].time := 3600.0, [91].log_data[21].valid := 1, [91].log_data[22].time := 3600.0, [91].log_data[22].valid := 1, [91].log_data[23].time := 3600.0, [91].log_data[23].valid := 1, [91].log_data[24].time := 3600.0, [91].log_data[24].valid := 1, [91].log_data[25].time := 3600.0, [91].log_data[25].valid := 1, [91].log_data[26].time := 3600.0, [91].log_data[26].valid := 1, [91].log_data[27].time := 3600.0, [91].log_data[27].valid := 1, [91].log_data[28].time := 3600.0, [91].log_data[28].valid := 1, [91].log_data[29].min := 1.0, [91].log_data[29].max := 1.0, [91].log_data[29].total := 3600.0, [91].log_data[29].time := 3600.0, [91].log_data[29].valid := 1, [91].log_data[30].min := 1.0, [91].log_data[30].max := 1.0, [91].log_data[30].total := 3600.0, [91].log_data[30].time := 3600.0, [91].log_data[30].valid := 1, [91].log_data[31].max := 1.0, [91].log_data[31].total := 1629.998, [91].log_data[31].time := 3600.0, [91].log_data[31].maxminute := 2, [91].log_data[31].valid := 1, [91].log_data[32].max := 1.0, [91].log_data[32].total := 1440.2471, [91].log_data[32].time := 3600.0, [91].log_data[32].minminute := 1, [91].log_data[32].valid := 1, [91].log_data[33].time := 3600.0, [91].log_data[33].valid := 1, [91].log_data[34].time := 3600.0, [91].log_data[34].valid := 1, [91].log_data[35].max := 1.0, [91].log_data[35].total := 1629.498, [91].log_data[35].time := 3600.0, [91].log_data[35].maxminute := 6, [91].log_data[35].valid := 1, [91].log_data[36].max := 1.0, [91].log_data[36].total := 1440.998, [91].log_data[36].time := 3600.0, [91].log_data[36].minminute := 5, [91].log_data[36].valid := 1,
        [91].log_data[37].max := 7.5991583, [91].log_data[37].total := 3625.4612, [91].log_data[37].time := 3600.0, [91].log_data[37].maxminute := 21, [91].log_data[37].valid := 1, [91].log_data[38].time := 3600.0, [91].log_data[38].valid := 1, [91].log_data[39].min := 0.9938818, [91].log_data[39].max := 1.0223833, [91].log_data[39].total := 3605.995, [91].log_data[39].time := 3600.0, [91].log_data[39].minminute := 45, [91].log_data[39].maxminute := 21, [91].log_data[39].valid := 1, [91].log_data[40].min := 7.5945454, [91].log_data[40].max := 7.60224, [91].log_data[40].total := 27354.176, [91].log_data[40].time := 3600.0, [91].log_data[40].minminute := 43, [91].log_data[40].maxminute := 2, [91].log_data[40].valid := 1, [91].log_data[41].min := 0.022540038, [91].log_data[41].max := 0.028232668, [91].log_data[41].total := 85.37348, [91].log_data[41].time := 3600.0, [91].log_data[41].minminute := 54, [91].log_data[41].maxminute := 34, [91].log_data[41].valid := 1, [91].log_data[42].min := 2.2916427, [91].log_data[42].max := 2.296236, [91].log_data[42].total := 8259.368, [91].log_data[42].time := 3600.0, [91].log_data[42].minminute := 41, [91].log_data[42].maxminute := 40, [91].log_data[42].valid := 1, [91].log_data[43].min := -0.27999878, [91].log_data[43].max := -0.26000214, [91].log_data[43].total := -1007.2925, [91].log_data[43].time := 3600.0, [91].log_data[43].valid := 1, [91].log_data[44].min := -0.3199997, [91].log_data[44].max := -0.30000305, [91].log_data[44].total := -1080.7054, [91].log_data[44].time := 3600.0, [91].log_data[44].valid := 1, [91].log_data[45].time := 3600.0, [91].log_data[45].valid := 1, [91].log_data[46].time := 3600.0, [91].log_data[46].valid := 1, [91].log_data[47].time := 3600.0, [91].log_data[47].valid := 1, [91].log_data[48].min := 6.5821533, [91].log_data[48].max := 6.9608383, [91].log_data[48].total := 24226.82, [91].log_data[48].time := 3600.0, [91].log_data[48].minminute := 52, [91].log_data[48].maxminute := 28, [91].log_data[48].valid := 1, [91].log_data[49].min := 6.911779, [91].log_data[49].max := 9.566228,
        [91].log_data[49].total := 29758.846, [91].log_data[49].time := 3600.0, [91].log_data[49].minminute := 48, [91].log_data[49].maxminute := 21, [91].log_data[49].valid := 1, [91].log_data[50].min := 2.0549152, [91].log_data[50].max := 2.1656237, [91].log_data[50].total := 7622.089, [91].log_data[50].time := 3600.0, [91].log_data[50].minminute := 21, [91].log_data[50].maxminute := 28, [91].log_data[50].valid := 1, [91].log_data[51].time := 3600.0, [91].log_data[51].valid := 1, [91].log_data[52].min := -2.9800034, [91].log_data[52].max := 0.11999512, [91].log_data[52].total := -7618.994, [91].log_data[52].time := 3600.0, [91].log_data[52].minminute := 23, [91].log_data[52].maxminute := 1, [91].log_data[52].valid := 1, [91].log_data[53].min := -2.4800034, [91].log_data[53].max := 0.27999878, [91].log_data[53].total := -6998.2236, [91].log_data[53].time := 3600.0, [91].log_data[53].minminute := 3, [91].log_data[53].maxminute := 26, [91].log_data[53].valid := 1, [91].log_data[54].max := 0.5415, [91].log_data[54].total := 1217.1797, [91].log_data[54].time := 3600.0, [91].log_data[54].minminute := 1, [91].log_data[54].maxminute := 23, [91].log_data[54].valid := 1, [91].log_data[55].max := 0.5655, [91].log_data[55].total := 1217.2465, [91].log_data[55].time := 3600.0, [91].log_data[55].minminute := 5, [91].log_data[55].maxminute := 27, [91].log_data[55].valid := 1, [91].log_data[56].min := 0.15977451, [91].log_data[56].max := 0.16024561, [91].log_data[56].total := 575.95416, [91].log_data[56].time := 3600.0, [91].log_data[56].minminute := 55, [91].log_data[56].maxminute := 3, [91].log_data[56].valid := 1, [91].log_data[57].min := 0.23911548, [91].log_data[57].max := 0.24084286, [91].log_data[57].total := 865.79565, [91].log_data[57].time := 3600.0, [91].log_data[57].minminute := 59, [91].log_data[57].maxminute := 2, [91].log_data[57].valid := 1, [91].log_data[58].time := 3600.0, [91].log_data[58].valid := 1, [91].log_data[59].time := 3600.0, [91].log_data[59].valid := 1, [91].log_data[60].valid := 1, [91].log_data[61].valid := 1,
        [91].log_data[62].valid := 1, [91].log_data[63].valid := 1, [91].log_data[64].valid := 1, [91].log_data[65].valid := 1, [91].log_data[66].valid := 1, [91].log_data[67].valid := 1, [91].log_data[68].valid := 1, [91].log_data[69].valid := 1, [91].log_data[70].valid := 1, [91].log_data[71].valid := 1, [91].log_data[72].valid := 1, [91].log_data[73].valid := 1, [91].log_data[74].valid := 1, [91].log_data[75].valid := 1, [91].log_data[76].valid := 1, [91].log_data[77].valid := 1, [91].log_data[78].valid := 1, [91].log_data[79].valid := 1, [91].log_data[80].valid := 1, [91].log_data[81].valid := 1, [91].log_data[82].valid := 1, [91].log_data[83].valid := 1, [91].log_data[84].valid := 1, [91].log_data[85].valid := 1, [91].log_data[86].valid := 1, [91].log_data[87].valid := 1, [91].log_data[88].valid := 1, [91].log_data[89].valid := 1, [91].log_data[90].valid := 1, [91].log_data[91].valid := 1, [91].log_data[92].valid := 1, [91].log_data[93].valid := 1, [91].log_data[94].valid := 1, [91].log_data[95].valid := 1, [91].log_data[96].valid := 1, [91].log_data[97].valid := 1, [91].log_data[98].valid := 1, [91].log_data[99].valid := 1, [91].log_data[100].valid := 1, [91].log_data[101].valid := 1, [91].log_data[102].valid := 1, [91].log_data[103].valid := 1, [91].log_data[104].valid := 1, [91].log_data[105].valid := 1, [91].log_data[106].valid := 1, [91].log_data[107].valid := 1, [91].log_data[108].valid := 1, [91].log_data[109].valid := 1, [91].log_data[110].valid := 1, [91].log_data[111].valid := 1, [91].log_data[112].valid := 1, [91].log_data[113].valid := 1, [91].log_data[114].valid := 1, [91].log_data[115].valid := 1, [91].log_data[116].valid := 1, [91].log_data[117].valid := 1, [91].log_data[118].valid := 1, [91].log_data[119].valid := 1, [91].log_data[120].valid := 1, [91].log_data[121].valid := 1,
        [91].log_data[122].valid := 1, [91].log_data[123].valid := 1, [91].log_data[124].valid := 1, [91].time.Year := 2023, [91].time.Month := 1, [91].time.Day := 16, [91].time.Hour := 22, [91].time.Minute := 59, [91].time.Second := 59, [92].log_data[0].min := 1.0, [92].log_data[0].max := 1.0, [92].log_data[0].total := 3600.0, [92].log_data[0].time := 3600.0, [92].log_data[0].valid := 1, [92].log_data[1].max := 1.0, [92].log_data[1].total := 472.249, [92].log_data[1].time := 3600.0, [92].log_data[1].maxminute := 52, [92].log_data[1].valid := 1, [92].log_data[2].max := 1.0, [92].log_data[2].total := 468.749, [92].log_data[2].time := 3600.0, [92].log_data[2].maxminute := 52, [92].log_data[2].valid := 1, [92].log_data[3].time := 3600.0, [92].log_data[3].valid := 1, [92].log_data[4].time := 3600.0, [92].log_data[4].valid := 1, [92].log_data[5].max := 1.0, [92].log_data[5].total := 161.249, [92].log_data[5].time := 3600.0, [92].log_data[5].maxminute := 54, [92].log_data[5].valid := 1, [92].log_data[6].time := 3600.0, [92].log_data[6].valid := 1, [92].log_data[7].time := 3600.0, [92].log_data[7].valid := 1, [92].log_data[8].min := 1.0, [92].log_data[8].max := 1.0, [92].log_data[8].total := 3600.0, [92].log_data[8].time := 3600.0, [92].log_data[8].valid := 1, [92].log_data[9].min := 1.0, [92].log_data[9].max := 1.0, [92].log_data[9].total := 3600.0, [92].log_data[9].time := 3600.0, [92].log_data[9].valid := 1, [92].log_data[10].min := 1.0, [92].log_data[10].max := 1.0, [92].log_data[10].total := 3600.0, [92].log_data[10].time := 3600.0, [92].log_data[10].valid := 1, [92].log_data[11].time := 3600.0, [92].log_data[11].valid := 1, [92].log_data[12].min := 1.0, [92].log_data[12].max := 1.0, [92].log_data[12].total := 3600.0, [92].log_data[12].time := 3600.0, [92].log_data[12].valid := 1, [92].log_data[13].min := 1.0,
        [92].log_data[13].max := 1.0, [92].log_data[13].total := 3600.0, [92].log_data[13].time := 3600.0, [92].log_data[13].valid := 1, [92].log_data[14].time := 3600.0, [92].log_data[14].valid := 1, [92].log_data[15].time := 3600.0, [92].log_data[15].valid := 1, [92].log_data[16].time := 3600.0, [92].log_data[16].valid := 1, [92].log_data[17].min := 1.0, [92].log_data[17].max := 1.0, [92].log_data[17].total := 3600.0, [92].log_data[17].time := 3600.0, [92].log_data[17].valid := 1, [92].log_data[18].time := 3600.0, [92].log_data[18].valid := 1, [92].log_data[19].time := 3600.0, [92].log_data[19].valid := 1, [92].log_data[20].time := 3600.0, [92].log_data[20].valid := 1, [92].log_data[21].min := 1.0, [92].log_data[21].max := 1.0, [92].log_data[21].total := 3600.0, [92].log_data[21].time := 3600.0, [92].log_data[21].valid := 1, [92].log_data[22].time := 3600.0, [92].log_data[22].valid := 1, [92].log_data[23].time := 3600.0, [92].log_data[23].valid := 1, [92].log_data[24].time := 3600.0, [92].log_data[24].valid := 1, [92].log_data[25].time := 3600.0, [92].log_data[25].valid := 1, [92].log_data[26].time := 3600.0, [92].log_data[26].valid := 1, [92].log_data[27].time := 3600.0, [92].log_data[27].valid := 1, [92].log_data[28].time := 3600.0, [92].log_data[28].valid := 1, [92].log_data[29].min := 1.0, [92].log_data[29].max := 1.0, [92].log_data[29].total := 3600.0, [92].log_data[29].time := 3600.0, [92].log_data[29].valid := 1, [92].log_data[30].min := 1.0, [92].log_data[30].max := 1.0, [92].log_data[30].total := 3600.0, [92].log_data[30].time := 3600.0, [92].log_data[30].valid := 1, [92].log_data[31].max := 1.0, [92].log_data[31].total := 1629.7471, [92].log_data[31].time := 3600.0, [92].log_data[31].maxminute := 5, [92].log_data[31].valid := 1, [92].log_data[32].max := 1.0, [92].log_data[32].total := 1440.998, [92].log_data[32].time := 3600.0, [92].log_data[32].minminute := 4, [92].log_data[32].valid := 1,
        [92].log_data[33].time := 3600.0, [92].log_data[33].valid := 1, [92].log_data[34].time := 3600.0, [92].log_data[34].valid := 1, [92].log_data[35].max := 1.0, [92].log_data[35].total := 1562.2471, [92].log_data[35].time := 3600.0, [92].log_data[35].maxminute := 9, [92].log_data[35].valid := 1, [92].log_data[36].max := 1.0, [92].log_data[36].total := 1596.749, [92].log_data[36].time := 3600.0, [92].log_data[36].minminute := 8, [92].log_data[36].valid := 1, [92].log_data[37].max := 7.3573275, [92].log_data[37].total := 3415.6306, [92].log_data[37].time := 3600.0, [92].log_data[37].maxminute := 53, [92].log_data[37].valid := 1, [92].log_data[38].time := 3600.0, [92].log_data[38].valid := 1, [92].log_data[39].min := 0.99293965, [92].log_data[39].max := 1.0233254, [92].log_data[39].total := 3601.886, [92].log_data[39].time := 3600.0, [92].log_data[39].minminute := 17, [92].log_data[39].maxminute := 59, [92].log_data[39].valid := 1, [92].log_data[40].min := 7.591798, [92].log_data[40].max := 7.603614, [92].log_data[40].total := 27352.873, [92].log_data[40].time := 3600.0, [92].log_data[40].minminute := 38, [92].log_data[40].maxminute := 46, [92].log_data[40].valid := 1, [92].log_data[41].min := 0.02273633, [92].log_data[41].max := 0.026073486, [92].log_data[41].total := 83.53369, [92].log_data[41].time := 3600.0, [92].log_data[41].maxminute := 9, [92].log_data[41].valid := 1, [92].log_data[42].min := 2.2916427, [92].log_data[42].max := 2.2964714, [92].log_data[42].total := 8259.372, [92].log_data[42].time := 3600.0, [92].log_data[42].minminute := 31, [92].log_data[42].maxminute := 47, [92].log_data[42].valid := 1, [92].log_data[43].min := -0.27999878, [92].log_data[43].max := -0.26000214, [92].log_data[43].total := -1006.4439, [92].log_data[43].time := 3600.0, [92].log_data[43].valid := 1, [92].log_data[44].min := -0.3199997, [92].log_data[44].max := -0.30000305, [92].log_data[44].total := -1080.2257, [92].log_data[44].time := 3600.0, [92].log_data[44].minminute := 8, [92].log_data[44].valid := 1, [92].log_data[45].time := 3600.0,
